  MoveL 5719 to (502.61, 490.4, 12.5) mm, rotated rx 0 ry 90 rz 0 deg; joints [-11.079, -27.597, 111.319, -15.089, -83.075, 50.859]
  Call Extruder(0.203)
  MoveL 5720 to (509.6, 490.4, 12.5) mm, rotated rx 0 ry 90 rz 0 deg; joints [-10.955, -27.463, 110.479, -14.987, -82.389, 51.03]
  Call Extruder(0.176)
  MoveL 5721 to (509.6, 496.43, 12.5) mm, rotated rx 0 ry 90 rz 0 deg; joints [-11.502, -27.439, 110.334, -15.543, -82.29, 51.128]
  Call Extruder(0.056)
  MoveL 5722 to (507.67, 496.44, 12.5) mm, rotated rx 0 ry 90 rz 0 deg; joints [-11.538, -27.477, 110.567, -15.572, -82.478, 51.079]
  Call Extruder(0.062)
  MoveL 5723 to (507.67, 498.58, 12.5) mm, rotated rx 0 ry 90 rz 0 deg; joints [-11.732, -27.468, 110.514, -15.77, -82.442, 51.114]
  Call Extruder(0.010)
  MoveL 5724 to (507.67, 498.93, 12.5) mm, rotated rx 0 ry 90 rz 0 deg; joints [-11.764, -27.467, 110.505, -15.802, -82.436, 51.12]
  Call Extruder(0.007)
  MoveL 5725 to (508.02, 498.93, 12.5) mm, rotated rx 0 ry 90 rz 0 deg; joints [-11.757, -27.46, 110.463, -15.797, -82.402, 51.129]
  Call Extruder(0.036)
  MoveL 5726 to (509.25, 498.93, 12.5) mm, rotated rx 0 ry 90 rz 0 deg; joints [-11.734, -27.436, 110.315, -15.778, -82.282, 51.16]
  Call Extruder(0.010)
  MoveL 5727 to (509.6, 498.93, 12.5) mm, rotated rx 0 ry 90 rz 0 deg; joints [-11.727, -27.429, 110.272, -15.772, -82.248, 51.169]
  Call Extruder(0.007)
  MoveL 5728 to (509.6, 499.28, 12.5) mm, rotated rx 0 ry 90 rz 0 deg; joints [-11.759, -27.427, 110.264, -15.805, -82.242, 51.175]
  Call Extruder(0.016)
  MoveL 5729 to (509.6, 499.84, 12.5) mm, rotated rx 0 ry 90 rz 0 deg; joints [-11.81, -27.425, 110.249, -15.856, -82.232, 51.184]
  Call Extruder(0.010)
  MoveL 5730 to (509.6, 500.19, 12.5) mm, rotated rx 0 ry 90 rz 0 deg; joints [-11.842, -27.423, 110.241, -15.889, -82.226, 51.19]
  Call Extruder(0.007)
  MoveL 5731 to (509.25, 500.19, 12.5) mm, rotated rx 0 ry 90 rz 0 deg; joints [-11.848, -27.43, 110.283, -15.894, -82.26, 51.181]
  Call Extruder(0.036)
  MoveL 5732 to (508.02, 500.19, 12.5) mm, rotated rx 0 ry 90 rz 0 deg; joints [-11.871, -27.455, 110.431, -15.913, -82.38, 51.149]
  Call Extruder(0.010)
  MoveL 5733 to (507.67, 500.19, 12.5) mm, rotated rx 0 ry 90 rz 0 deg; joints [-11.878, -27.462, 110.473, -15.918, -82.414, 51.141]
  Call Extruder(0.007)
  MoveL 5734 to (507.67, 500.54, 12.5) mm, rotated rx 0 ry 90 rz 0 deg; joints [-11.91, -27.46, 110.464, -15.95, -82.408, 51.146]
  Call Extruder(0.062)
  MoveL 5735 to (507.67, 502.67, 12.5) mm, rotated rx 0 ry 90 rz 0 deg; joints [-12.103, -27.451, 110.41, -16.147, -82.371, 51.182]
  Call Extruder(0.056)
  MoveL 5736 to (509.6, 502.68, 12.5) mm, rotated rx 0 ry 90 rz 0 deg; joints [-12.066, -27.413, 110.177, -16.116, -82.183, 51.232]
  Call Extruder(0.202)
  MoveL 5737 to (509.6, 509.6, 12.5) mm, rotated rx 0 ry 90 rz 0 deg; joints [-12.688, -27.382, 109.994, -16.751, -82.06, 51.352]
  Call Extruder(0.559)
  MoveL 5738 to (490.4, 509.6, 12.5) mm, rotated rx 0 ry 90 rz 0 deg; joints [-13.088, -27.741, 112.282, -17.084, -83.918, 50.83]
  MoveL 5739 to (490.4, 490.4, 12.5) mm, rotated rx 0 ry 90 rz 0 deg; joints [-11.303, -27.811, 112.772, -15.278, -84.276, 50.554]
  Call Extruder(0.177)
  MoveL 5740 to (496.5, 490.4, 12.5) mm, rotated rx 0 ry 90 rz 0 deg; joints [-11.19, -27.707, 112.049, -15.182, -83.676, 50.708]
  Call Extruder(0.010)
  MoveL 5741 to (496.85, 490.4, 12.5) mm, rotated rx 0 ry 90 rz 0 deg; joints [-11.184, -27.701, 112.007, -15.177, -83.641, 50.717]
  Call Extruder(0.007)
  MoveL 5742 to (496.85, 490.75, 12.5) mm, rotated rx 0 ry 90 rz 0 deg; joints [-11.216, -27.7, 111.999, -15.209, -83.635, 50.721]
  Call Extruder(0.035)
  MoveL 5743 to (496.84, 491.95, 12.5) mm, rotated rx 0 ry 90 rz 0 deg; joints [-11.327, -27.696, 111.971, -15.322, -83.615, 50.739]
  Call Extruder(0.010)
  MoveL 5744 to (496.84, 492.3, 12.5) mm, rotated rx 0 ry 90 rz 0 deg; joints [-11.36, -27.694, 111.962, -15.355, -83.609, 50.744]
  Call Extruder(0.007)
  MoveL 5745 to (497.19, 492.3, 12.5) mm, rotated rx 0 ry 90 rz 0 deg; joints [-11.353, -27.688, 111.921, -15.349, -83.575, 50.752]
  Call Extruder(0.061)
  MoveL 5746 to (499.3, 492.3, 12.5) mm, rotated rx 0 ry 90 rz 0 deg; joints [-11.314, -27.65, 111.669, -15.316, -83.367, 50.805]
  Call Extruder(0.055)
  MoveL 5747 to (499.3, 490.4, 12.5) mm, rotated rx 0 ry 90 rz 0 deg; joints [-11.139, -27.657, 111.714, -15.139, -83.399, 50.778]
  Call Extruder(0.016)
  MoveL 5748 to (499.84, 490.4, 12.5) mm, rotated rx 0 ry 90 rz 0 deg; joints [-11.129, -27.648, 111.65, -15.131, -83.347, 50.791]
  Call Extruder(0.042)
  MoveL 5749 to (499.84, 492.3, 12.5) mm, rotated rx 0 ry 90 rz 0 deg; joints [-11.304, -27.641, 111.605, -15.308, -83.315, 50.819]
  Call Extruder(0.060)
  MoveL 5750 to (501.91, 492.3, 12.5) mm, rotated rx 0 ry 90 rz 0 deg; joints [-11.266, -27.603, 111.358, -15.276, -83.112, 50.871]
  Call Extruder(0.007)
  MoveL 5751 to (502.26, 492.3, 12.5) mm, rotated rx 0 ry 90 rz 0 deg; joints [-11.26, -27.596, 111.316, -15.271, -83.077, 50.879]
  Set speed (120.0 mm/s)
  MoveL 5752 to (502.26, 491.95, 12.5) mm, rotated rx 0 ry 90 rz 0 deg; joints [-11.228, -27.598, 111.324, -15.238, -83.083, 50.874]
  Set speed (1000.0 mm/s)
  MoveL 5753 to (502.26, 491.9, 12.5) mm, rotated rx 0 ry 90 rz 0 deg; joints [-11.223, -27.598, 111.325, -15.234, -83.084, 50.873]
  Set speed (1000.0 mm/s)
  MoveL 5754 to (502.36, 491.9, 12.5) mm, rotated rx 0 ry 90 rz 0 deg; joints [-11.221, -27.596, 111.313, -15.232, -83.074, 50.876]
  Set speed (1000.0 mm/s)
  MoveL 5755 to (507.28, 499.36, 12.5) mm, rotated rx 0 ry 90 rz 0 deg; joints [-11.811, -27.473, 110.54, -15.848, -82.466, 51.117]
  Set speed (1000.0 mm/s)
  MoveL 5756 to (507.53, 499.61, 12.5) mm, rotated rx 0 ry 90 rz 0 deg; joints [-11.828, -27.467, 110.505, -15.867, -82.438, 51.127]
  Set speed (15.0 mm/s)
  Call Extruder(0.014)
  MoveL 5757 to (507.97, 499.56, 12.5) mm, rotated rx 0 ry 90 rz 0 deg; joints [-11.815, -27.458, 110.452, -15.855, -82.396, 51.138]
  Call Extruder(0.030)
  MoveL 5758 to (508.96, 499.56, 12.5) mm, rotated rx 0 ry 90 rz 0 deg; joints [-11.796, -27.439, 110.333, -15.84, -82.299, 51.163]
  Call Extruder(0.011)
  MoveL 5759 to (509.21, 499.31, 12.5) mm, rotated rx 0 ry 90 rz 0 deg; joints [-11.77, -27.435, 110.309, -15.814, -82.279, 51.165]
  Set speed (120.0 mm/s)
  MoveL 5760 to (508.9, 499.63, 12.5) mm, rotated rx 0 ry 90 rz 0 deg; joints [-11.804, -27.44, 110.339, -15.848, -82.304, 51.163]
  Set speed (1000.0 mm/s)
  MoveL 5761 to (490.68, 490.68, 12.5) mm, rotated rx 0 ry 90 rz 0 deg; joints [-11.324, -27.805, 112.732, -15.3, -84.244, 50.565]
  Set speed (1000.0 mm/s)
  MoveL 5762 to (490.68, 490.68, 12.6) mm, rotated rx 0 ry 90 rz 0 deg; joints [-11.324, -27.816, 112.737, -15.3, -84.238, 50.567]
  Set speed (30.0 mm/s)
  Call Extruder(0.767)
  MoveL 5763 to (509.32, 509.32, 12.6) mm, rotated rx 0 ry 90 rz 0 deg; joints [-12.669, -27.4, 110.041, -16.73, -82.087, 51.341]
  MoveL 5764 to (509.44, 509.44, 12.6) mm, rotated rx 0 ry 90 rz 0 deg; joints [-12.677, -27.397, 110.023, -16.739, -82.073, 51.347]
  Set speed (120.0 mm/s)
  MoveL 5765 to (507.39, 502.51, 12.6) mm, rotated rx 0 ry 90 rz 0 deg; joints [-12.094, -27.468, 110.453, -16.137, -82.396, 51.173]
  Set speed (30.0 mm/s)
  Call Extruder(0.280)
  MoveL 5766 to (500.58, 509.32, 12.6) mm, rotated rx 0 ry 90 rz 0 deg; joints [-12.847, -27.57, 111.088, -16.877, -82.932, 51.106]
  Set speed (120.0 mm/s)
  MoveL 5767 to (499.42, 509.32, 12.6) mm, rotated rx 0 ry 90 rz 0 deg; joints [-12.872, -27.592, 111.226, -16.897, -83.044, 51.075]
  Set speed (30.0 mm/s)
  Call Extruder(0.360)
  MoveL 5768 to (490.68, 500.58, 12.6) mm, rotated rx 0 ry 90 rz 0 deg; joints [-12.247, -27.781, 112.493, -16.233, -84.059, 50.705]
  Set speed (120.0 mm/s)
  MoveL 5769 to (490.68, 499.42, 12.6) mm, rotated rx 0 ry 90 rz 0 deg; joints [-12.139, -27.786, 112.523, -16.124, -84.081, 50.688]
  Set speed (30.0 mm/s)
  Call Extruder(0.282)
  MoveL 5770 to (497.52, 492.58, 12.6) mm, rotated rx 0 ry 90 rz 0 deg; joints [-11.373, -27.692, 111.88, -15.37, -83.533, 50.766]
  MoveL 5771 to (497.64, 492.46, 12.6) mm, rotated rx 0 ry 90 rz 0 deg; joints [-11.359, -27.69, 111.869, -15.357, -83.523, 50.767]
  Set speed (120.0 mm/s)
  MoveL 5772 to (502.48, 492.58, 12.6) mm, rotated rx 0 ry 90 rz 0 deg; joints [-11.281, -27.602, 111.288, -15.294, -83.046, 50.89]
  Set speed (30.0 mm/s)
  Call Extruder(0.202)
  MoveL 5773 to (507.39, 497.49, 12.6) mm, rotated rx 0 ry 90 rz 0 deg; joints [-11.639, -27.489, 110.58, -15.674, -82.483, 51.091]
  MoveL 5774 to (507.51, 497.61, 12.6) mm, rotated rx 0 ry 90 rz 0 deg; joints [-11.647, -27.486, 110.562, -15.683, -82.469, 51.096]
  Set speed (120.0 mm/s)
  MoveL 5775 to (509.32, 490.68, 12.6) mm, rotated rx 0 ry 90 rz 0 deg; joints [-10.985, -27.478, 110.511, -15.017, -82.407, 51.029]
  Set speed (30.0 mm/s)
  Call Extruder(0.767)
  MoveL 5776 to (490.68, 509.32, 12.6) mm, rotated rx 0 ry 90 rz 0 deg; joints [-13.056, -27.748, 112.262, -17.053, -83.891, 50.835]
  MoveL 5777 to (490.56, 509.44, 12.6) mm, rotated rx 0 ry 90 rz 0 deg; joints [-13.07, -27.75, 112.273, -17.067, -83.901, 50.833]
  Set speed (120.0 mm/s)
  MoveL 5778 to (496.72, 492.37, 12.6) mm, rotated rx 0 ry 90 rz 0 deg; joints [-11.369, -27.707, 111.981, -15.363, -83.615, 50.743]
  Set speed (1000.0 mm/s)
  MoveL 5779 to (496.79, 492.3, 12.6) mm, rotated rx 0 ry 90 rz 0 deg; joints [-11.361, -27.706, 111.974, -15.356, -83.609, 50.744]
  Set speed (15.0 mm/s)
  Call Extruder(0.072)
  MoveL 5780 to (499.25, 492.3, 12.6) mm, rotated rx 0 ry 90 rz 0 deg; joints [-11.315, -27.662, 111.681, -15.317, -83.368, 50.806]
  Call Extruder(0.055)
  MoveL 5781 to (499.25, 490.4, 12.6) mm, rotated rx 0 ry 90 rz 0 deg; joints [-11.14, -27.669, 111.726, -15.14, -83.4, 50.778]
  Call Extruder(0.019)
  MoveL 5782 to (499.9, 490.4, 12.6) mm, rotated rx 0 ry 90 rz 0 deg; joints [-11.128, -27.657, 111.648, -15.13, -83.336, 50.794]
  Call Extruder(0.052)
  MoveL 5783 to (499.9, 492.3, 12.6) mm, rotated rx 0 ry 90 rz 0 deg; joints [-11.303, -27.65, 111.603, -15.307, -83.303, 50.822]
  Call Extruder(0.060)
  MoveL 5784 to (501.97, 492.3, 12.6) mm, rotated rx 0 ry 90 rz 0 deg; joints [-11.265, -27.612, 111.355, -15.276, -83.1, 50.874]
  Call Extruder(0.010)
  MoveL 5785 to (502.32, 492.3, 12.6) mm, rotated rx 0 ry 90 rz 0 deg; joints [-11.259, -27.606, 111.313, -15.27, -83.066, 50.882]
  Call Extruder(0.007)
  MoveL 5786 to (502.32, 491.95, 12.6) mm, rotated rx 0 ry 90 rz 0 deg; joints [-11.227, -27.607, 111.322, -15.238, -83.072, 50.877]
  Call Extruder(0.035)
  MoveL 5787 to (502.32, 490.75, 12.6) mm, rotated rx 0 ry 90 rz 0 deg; joints [-11.116, -27.611, 111.35, -15.126, -83.092, 50.859]
  Call Extruder(0.010)
  MoveL 5788 to (502.32, 490.4, 12.6) mm, rotated rx 0 ry 90 rz 0 deg; joints [-11.084, -27.613, 111.358, -15.094, -83.098, 50.854]
  Call Extruder(0.007)
  MoveL 5789 to (502.67, 490.4, 12.6) mm, rotated rx 0 ry 90 rz 0 deg; joints [-11.078, -27.606, 111.317, -15.088, -83.063, 50.862]
  Call Extruder(0.202)
  MoveL 5790 to (509.6, 490.4, 12.6) mm, rotated rx 0 ry 90 rz 0 deg; joints [-10.955, -27.473, 110.484, -14.987, -82.384, 51.032]
  Call Extruder(0.174)
  MoveL 5791 to (509.6, 496.37, 12.6) mm, rotated rx 0 ry 90 rz 0 deg; joints [-11.496, -27.45, 110.341, -15.538, -82.286, 51.128]
  Call Extruder(0.056)
  MoveL 5792 to (507.67, 496.38, 12.6) mm, rotated rx 0 ry 90 rz 0 deg; joints [-11.532, -27.488, 110.573, -15.567, -82.474, 51.08]
  Call Extruder(0.073)
  MoveL 5793 to (507.67, 498.87, 12.6) mm, rotated rx 0 ry 90 rz 0 deg; joints [-11.759, -27.478, 110.511, -15.797, -82.432, 51.12]
  Call Extruder(0.056)
  MoveL 5794 to (509.6, 498.87, 12.6) mm, rotated rx 0 ry 90 rz 0 deg; joints [-11.722, -27.439, 110.279, -15.767, -82.244, 51.169]
  Call Extruder(0.030)
  MoveL 5795 to (509.6, 499.9, 12.6) mm, rotated rx 0 ry 90 rz 0 deg; joints [-11.815, -27.435, 110.253, -15.862, -82.226, 51.186]
  Call Extruder(0.010)
  MoveL 5796 to (509.6, 500.25, 12.6) mm, rotated rx 0 ry 90 rz 0 deg; joints [-11.847, -27.434, 110.244, -15.894, -82.22, 51.192]
  Call Extruder(0.007)
  MoveL 5797 to (509.25, 500.25, 12.6) mm, rotated rx 0 ry 90 rz 0 deg; joints [-11.853, -27.441, 110.286, -15.899, -82.254, 51.183]
  Call Extruder(0.036)
  MoveL 5798 to (508.02, 500.25, 12.6) mm, rotated rx 0 ry 90 rz 0 deg; joints [-11.876, -27.465, 110.435, -15.918, -82.374, 51.152]
  Call Extruder(0.010)
  MoveL 5799 to (507.67, 500.25, 12.6) mm, rotated rx 0 ry 90 rz 0 deg; joints [-11.883, -27.472, 110.477, -15.924, -82.408, 51.143]
  Call Extruder(0.007)
  MoveL 5800 to (507.67, 500.6, 12.6) mm, rotated rx 0 ry 90 rz 0 deg; joints [-11.915, -27.471, 110.468, -15.956, -82.402, 51.149]
  Call Extruder(0.062)
  MoveL 5801 to (507.67, 502.73, 12.6) mm, rotated rx 0 ry 90 rz 0 deg; joints [-12.108, -27.462, 110.414, -16.152, -82.365, 51.184]
  Call Extruder(0.056)
  MoveL 5802 to (509.6, 502.73, 12.6) mm, rotated rx 0 ry 90 rz 0 deg; joints [-12.071, -27.423, 110.181, -16.122, -82.177, 51.234]
  Call Extruder(0.200)
  MoveL 5803 to (509.6, 509.6, 12.6) mm, rotated rx 0 ry 90 rz 0 deg; joints [-12.688, -27.393, 109.999, -16.751, -82.055, 51.354]
  Call Extruder(0.559)
  MoveL 5804 to (490.4, 509.6, 12.6) mm, rotated rx 0 ry 90 rz 0 deg; joints [-13.088, -27.752, 112.287, -17.084, -83.913, 50.831]
  MoveL 5805 to (490.4, 490.4, 12.6) mm, rotated rx 0 ry 90 rz 0 deg; joints [-11.303, -27.821, 112.777, -15.278, -84.271, 50.556]
  Call Extruder(0.176)
  MoveL 5806 to (496.44, 490.4, 12.6) mm, rotated rx 0 ry 90 rz 0 deg; joints [-11.191, -27.719, 112.061, -15.183, -83.676, 50.708]
  Call Extruder(0.010)
  MoveL 5807 to (496.79, 490.4, 12.6) mm, rotated rx 0 ry 90 rz 0 deg; joints [-11.185, -27.713, 112.019, -15.178, -83.642, 50.717]
  Call Extruder(0.007)
  MoveL 5808 to (496.79, 490.75, 12.6) mm, rotated rx 0 ry 90 rz 0 deg; joints [-11.217, -27.711, 112.011, -15.21, -83.636, 50.722]
  Call Extruder(0.045)
  MoveL 5809 to (496.79, 492.3, 12.6) mm, rotated rx 0 ry 90 rz 0 deg; joints [-11.361, -27.706, 111.974, -15.356, -83.609, 50.744]
  Set speed (120.0 mm/s)
  MoveL 5810 to (497.19, 492.3, 12.6) mm, rotated rx 0 ry 90 rz 0 deg; joints [-11.353, -27.699, 111.926, -15.349, -83.57, 50.754]
  Set speed (1000.0 mm/s)
  MoveL 5811 to (497.19, 492.4, 12.6) mm, rotated rx 0 ry 90 rz 0 deg; joints [-11.363, -27.699, 111.924, -15.359, -83.568, 50.755]
  Set speed (1000.0 mm/s)
  MoveL 5812 to (507.28, 499.5, 12.6) mm, rotated rx 0 ry 90 rz 0 deg; joints [-11.822, -27.483, 110.542, -15.86, -82.459, 51.121]
  Set speed (15.0 mm/s)
  Call Extruder(0.006)
  MoveL 5813 to (507.58, 499.2, 12.6) mm, rotated rx 0 ry 90 rz 0 deg; joints [-11.79, -27.478, 110.514, -15.829, -82.435, 51.123]
  Set speed (120.0 mm/s)
  MoveL 5814 to (508.07, 499.2, 12.6) mm, rotated rx 0 ry 90 rz 0 deg; joints [-11.781, -27.468, 110.455, -15.821, -82.387, 51.136]
  Set speed (15.0 mm/s)
  Call Extruder(0.015)
  MoveL 5815 to (507.36, 499.91, 12.6) mm, rotated rx 0 ry 90 rz 0 deg; joints [-11.859, -27.48, 110.522, -15.898, -82.444, 51.13]
  Set speed (120.0 mm/s)
  MoveL 5816 to (507.85, 499.92, 12.6) mm, rotated rx 0 ry 90 rz 0 deg; joints [-11.85, -27.47, 110.463, -15.89, -82.396, 51.142]
  Set speed (15.0 mm/s)
  Call Extruder(0.015)
  MoveL 5817 to (508.57, 499.2, 12.6) mm, rotated rx 0 ry 90 rz 0 deg; joints [-11.771, -27.459, 110.395, -15.813, -82.339, 51.149]
  Set speed (120.0 mm/s)
  MoveL 5818 to (509.06, 499.2, 12.6) mm, rotated rx 0 ry 90 rz 0 deg; joints [-11.762, -27.449, 110.335, -15.806, -82.29, 51.161]
  Set speed (15.0 mm/s)
  Call Extruder(0.015)
  MoveL 5819 to (508.35, 499.92, 12.6) mm, rotated rx 0 ry 90 rz 0 deg; joints [-11.84, -27.46, 110.404, -15.883, -82.348, 51.155]
  Set speed (120.0 mm/s)
  MoveL 5820 to (508.84, 499.92, 12.6) mm, rotated rx 0 ry 90 rz 0 deg; joints [-11.831, -27.45, 110.344, -15.875, -82.3, 51.167]
  Set speed (15.0 mm/s)
  Call Extruder(0.009)
  MoveL 5821 to (509.27, 499.49, 12.6) mm, rotated rx 0 ry 90 rz 0 deg; joints [-11.784, -27.443, 110.303, -15.829, -82.266, 51.171]
  Set speed (120.0 mm/s)
  MoveL 5822 to (508.9, 499.57, 12.6) mm, rotated rx 0 ry 90 rz 0 deg; joints [-11.799, -27.45, 110.346, -15.842, -82.3, 51.163]
  Set speed (1000.0 mm/s)
  MoveL 5823 to (490.68, 490.68, 12.6) mm, rotated rx 0 ry 90 rz 0 deg; joints [-11.324, -27.816, 112.737, -15.3, -84.238, 50.567]
  Set speed (1000.0 mm/s)
  MoveL 5824 to (490.68, 490.68, 12.7) mm, rotated rx 0 ry 90 rz 0 deg; joints [-11.324, -27.826, 112.742, -15.3, -84.233, 50.568]
  Set speed (30.0 mm/s)
  Call Extruder(0.767)
  MoveL 5825 to (509.32, 509.32, 12.7) mm, rotated rx 0 ry 90 rz 0 deg; joints [-12.669, -27.41, 110.046, -16.73, -82.082, 51.343]
  MoveL 5826 to (509.44, 509.44, 12.7) mm, rotated rx 0 ry 90 rz 0 deg; joints [-12.677, -27.407, 110.028, -16.739, -82.068, 51.348]
  Set speed (120.0 mm/s)
  MoveL 5827 to (507.38, 502.51, 12.7) mm, rotated rx 0 ry 90 rz 0 deg; joints [-12.094, -27.479, 110.458, -16.137, -82.391, 51.175]
  Set speed (30.0 mm/s)
  Call Extruder(0.280)
  MoveL 5828 to (500.58, 509.32, 12.7) mm, rotated rx 0 ry 90 rz 0 deg; joints [-12.847, -27.581, 111.093, -16.877, -82.927, 51.108]
  Set speed (120.0 mm/s)
  MoveL 5829 to (499.42, 509.32, 12.7) mm, rotated rx 0 ry 90 rz 0 deg; joints [-12.872, -27.603, 111.231, -16.897, -83.039, 51.077]
  Set speed (30.0 mm/s)
  Call Extruder(0.360)
  MoveL 5830 to (490.68, 500.58, 12.7) mm, rotated rx 0 ry 90 rz 0 deg; joints [-12.247, -27.792, 112.498, -16.234, -84.054, 50.706]
  Set speed (120.0 mm/s)
  MoveL 5831 to (490.68, 499.42, 12.7) mm, rotated rx 0 ry 90 rz 0 deg; joints [-12.139, -27.796, 112.528, -16.124, -84.076, 50.689]
  Set speed (30.0 mm/s)
  Call Extruder(0.281)
  MoveL 5832 to (497.52, 492.58, 12.7) mm, rotated rx 0 ry 90 rz 0 deg; joints [-11.373, -27.703, 111.886, -15.371, -83.527, 50.768]
  MoveL 5833 to (497.64, 492.46, 12.7) mm, rotated rx 0 ry 90 rz 0 deg; joints [-11.359, -27.701, 111.874, -15.357, -83.517, 50.769]
  Set speed (120.0 mm/s)
  MoveL 5834 to (502.48, 492.58, 12.7) mm, rotated rx 0 ry 90 rz 0 deg; joints [-11.282, -27.612, 111.293, -15.294, -83.041, 50.892]
  Set speed (30.0 mm/s)
  Call Extruder(0.202)
  MoveL 5835 to (507.39, 497.49, 12.7) mm, rotated rx 0 ry 90 rz 0 deg; joints [-11.639, -27.499, 110.585, -15.674, -82.478, 51.092]
  MoveL 5836 to (507.51, 497.61, 12.7) mm, rotated rx 0 ry 90 rz 0 deg; joints [-11.647, -27.496, 110.567, -15.683, -82.464, 51.097]
  Set speed (120.0 mm/s)
  MoveL 5837 to (508.99, 499.09, 12.7) mm, rotated rx 0 ry 90 rz 0 deg; joints [-11.754, -27.461, 110.352, -15.797, -82.294, 51.159]
  Set speed (30.0 mm/s)
  Call Extruder(0.013)
  MoveL 5838 to (509.32, 499.42, 12.7) mm, rotated rx 0 ry 90 rz 0 deg; joints [-11.777, -27.453, 110.304, -15.822, -82.257, 51.173]
  Set speed (120.0 mm/s)
  MoveL 5839 to (507.64, 498.84, 12.7) mm, rotated rx 0 ry 90 rz 0 deg; joints [-11.756, -27.489, 110.521, -15.795, -82.43, 51.121]
  Set speed (1000.0 mm/s)
  MoveL 5840 to (507.64, 496.29, 12.7) mm, rotated rx 0 ry 90 rz 0 deg; joints [-11.525, -27.499, 110.584, -15.559, -82.473, 51.079]
  Set speed (1000.0 mm/s)
  MoveL 5841 to (509.32, 490.68, 12.7) mm, rotated rx 0 ry 90 rz 0 deg; joints [-10.985, -27.488, 110.516, -15.017, -82.402, 51.031]
  Set speed (30.0 mm/s)
  Call Extruder(0.767)
  MoveL 5842 to (490.68, 509.32, 12.7) mm, rotated rx 0 ry 90 rz 0 deg; joints [-13.056, -27.759, 112.267, -17.053, -83.886, 50.836]
  MoveL 5843 to (490.56, 509.44, 12.7) mm, rotated rx 0 ry 90 rz 0 deg; joints [-13.07, -27.76, 112.278, -17.067, -83.895, 50.835]
  Set speed (120.0 mm/s)
  MoveL 5844 to (502.46, 492.37, 12.7) mm, rotated rx 0 ry 90 rz 0 deg; joints [-11.263, -27.613, 111.301, -15.275, -83.046, 50.888]
  Set speed (1000.0 mm/s)
  MoveL 5845 to (502.39, 492.3, 12.7) mm, rotated rx 0 ry 90 rz 0 deg; joints [-11.257, -27.615, 111.311, -15.269, -83.054, 50.885]
  Set speed (15.0 mm/s)
  Call Extruder(0.010)
  MoveL 5846 to (502.39, 491.95, 12.7) mm, rotated rx 0 ry 90 rz 0 deg; joints [-11.225, -27.616, 111.319, -15.237, -83.06, 50.88]
  Call Extruder(0.035)
  MoveL 5847 to (502.39, 490.75, 12.7) mm, rotated rx 0 ry 90 rz 0 deg; joints [-11.115, -27.621, 111.348, -15.125, -83.08, 50.862]
  Call Extruder(0.010)
  MoveL 5848 to (502.39, 490.4, 12.7) mm, rotated rx 0 ry 90 rz 0 deg; joints [-11.083, -27.622, 111.356, -15.093, -83.086, 50.857]
  Call Extruder(0.007)
  MoveL 5849 to (502.74, 490.4, 12.7) mm, rotated rx 0 ry 90 rz 0 deg; joints [-11.077, -27.616, 111.314, -15.088, -83.052, 50.865]
  Call Extruder(0.200)
  MoveL 5850 to (509.6, 490.4, 12.7) mm, rotated rx 0 ry 90 rz 0 deg; joints [-10.955, -27.484, 110.489, -14.988, -82.378, 51.033]
  Call Extruder(0.172)
  MoveL 5851 to (509.6, 496.31, 12.7) mm, rotated rx 0 ry 90 rz 0 deg; joints [-11.491, -27.46, 110.347, -15.532, -82.282, 51.128]
  Call Extruder(0.056)
  MoveL 5852 to (507.67, 496.31, 12.7) mm, rotated rx 0 ry 90 rz 0 deg; joints [-11.527, -27.499, 110.58, -15.562, -82.47, 51.08]
  Call Extruder(0.062)
  MoveL 5853 to (507.67, 498.46, 12.7) mm, rotated rx 0 ry 90 rz 0 deg; joints [-11.722, -27.49, 110.527, -15.759, -82.434, 51.115]
  Call Extruder(0.010)
  MoveL 5854 to (507.67, 498.81, 12.7) mm, rotated rx 0 ry 90 rz 0 deg; joints [-11.753, -27.488, 110.518, -15.792, -82.428, 51.121]
  Call Extruder(0.007)
  MoveL 5855 to (508.02, 498.81, 12.7) mm, rotated rx 0 ry 90 rz 0 deg; joints [-11.747, -27.482, 110.476, -15.786, -82.394, 51.13]
  Call Extruder(0.036)
  MoveL 5856 to (509.25, 498.81, 12.7) mm, rotated rx 0 ry 90 rz 0 deg; joints [-11.723, -27.457, 110.328, -15.767, -82.274, 51.161]
  Call Extruder(0.010)
  MoveL 5857 to (509.6, 498.81, 12.7) mm, rotated rx 0 ry 90 rz 0 deg; joints [-11.717, -27.45, 110.286, -15.762, -82.24, 51.17]
  Call Extruder(0.007)
  MoveL 5858 to (509.6, 499.16, 12.7) mm, rotated rx 0 ry 90 rz 0 deg; joints [-11.749, -27.449, 110.277, -15.794, -82.234, 51.176]
  Call Extruder(0.023)
  MoveL 5859 to (509.6, 499.95, 12.7) mm, rotated rx 0 ry 90 rz 0 deg; joints [-11.82, -27.445, 110.257, -15.867, -82.22, 51.189]
  Call Extruder(0.010)
  MoveL 5860 to (509.6, 500.3, 12.7) mm, rotated rx 0 ry 90 rz 0 deg; joints [-11.852, -27.444, 110.248, -15.899, -82.214, 51.195]
  Call Extruder(0.007)
  MoveL 5861 to (509.25, 500.3, 12.7) mm, rotated rx 0 ry 90 rz 0 deg; joints [-11.858, -27.451, 110.29, -15.905, -82.248, 51.186]
  Call Extruder(0.036)
  MoveL 5862 to (508.02, 500.3, 12.7) mm, rotated rx 0 ry 90 rz 0 deg; joints [-11.882, -27.475, 110.439, -15.924, -82.368, 51.154]
  Call Extruder(0.010)
  MoveL 5863 to (507.67, 500.3, 12.7) mm, rotated rx 0 ry 90 rz 0 deg; joints [-11.888, -27.482, 110.481, -15.929, -82.402, 51.145]
  Call Extruder(0.007)
  MoveL 5864 to (507.67, 500.65, 12.7) mm, rotated rx 0 ry 90 rz 0 deg; joints [-11.92, -27.481, 110.472, -15.961, -82.396, 51.151]
  Call Extruder(0.062)
  MoveL 5865 to (507.67, 502.79, 12.7) mm, rotated rx 0 ry 90 rz 0 deg; joints [-12.113, -27.472, 110.417, -16.157, -82.359, 51.187]
  Call Extruder(0.056)
  MoveL 5866 to (509.6, 502.79, 12.7) mm, rotated rx 0 ry 90 rz 0 deg; joints [-12.076, -27.433, 110.185, -16.127, -82.171, 51.237]
  Call Extruder(0.198)
  MoveL 5867 to (509.6, 509.6, 12.7) mm, rotated rx 0 ry 90 rz 0 deg; joints [-12.688, -27.403, 110.004, -16.751, -82.049, 51.355]
  Call Extruder(0.559)
  MoveL 5868 to (490.4, 509.6, 12.7) mm, rotated rx 0 ry 90 rz 0 deg; joints [-13.088, -27.762, 112.292, -17.084, -83.907, 50.833]
  MoveL 5869 to (490.4, 490.4, 12.7) mm, rotated rx 0 ry 90 rz 0 deg; joints [-11.303, -27.832, 112.782, -15.279, -84.265, 50.557]
  Call Extruder(0.174)
  MoveL 5870 to (496.38, 490.4, 12.7) mm, rotated rx 0 ry 90 rz 0 deg; joints [-11.192, -27.73, 112.072, -15.184, -83.676, 50.708]
  Call Extruder(0.010)
  MoveL 5871 to (496.73, 490.4, 12.7) mm, rotated rx 0 ry 90 rz 0 deg; joints [-11.186, -27.724, 112.031, -15.179, -83.642, 50.717]
  Call Extruder(0.007)
  MoveL 5872 to (496.73, 490.75, 12.7) mm, rotated rx 0 ry 90 rz 0 deg; joints [-11.218, -27.723, 112.023, -15.211, -83.636, 50.722]
  Call Extruder(0.035)
  MoveL 5873 to (496.73, 491.95, 12.7) mm, rotated rx 0 ry 90 rz 0 deg; joints [-11.329, -27.719, 111.994, -15.324, -83.615, 50.739]
  Call Extruder(0.010)
  MoveL 5874 to (496.73, 492.3, 12.7) mm, rotated rx 0 ry 90 rz 0 deg; joints [-11.362, -27.718, 111.986, -15.357, -83.609, 50.744]
  Call Extruder(0.007)
  MoveL 5875 to (497.08, 492.3, 12.7) mm, rotated rx 0 ry 90 rz 0 deg; joints [-11.355, -27.711, 111.944, -15.351, -83.575, 50.753]
  Call Extruder(0.061)
  MoveL 5876 to (499.19, 492.3, 12.7) mm, rotated rx 0 ry 90 rz 0 deg; joints [-11.316, -27.674, 111.693, -15.318, -83.368, 50.806]
  Call Extruder(0.055)
  MoveL 5877 to (499.19, 490.4, 12.7) mm, rotated rx 0 ry 90 rz 0 deg; joints [-11.141, -27.68, 111.738, -15.141, -83.4, 50.778]
  Call Extruder(0.022)
  MoveL 5878 to (499.96, 490.4, 12.7) mm, rotated rx 0 ry 90 rz 0 deg; joints [-11.127, -27.666, 111.646, -15.129, -83.324, 50.797]
  Call Extruder(0.055)
  MoveL 5879 to (499.97, 492.3, 12.7) mm, rotated rx 0 ry 90 rz 0 deg; joints [-11.302, -27.66, 111.6, -15.307, -83.292, 50.825]
  Call Extruder(0.060)
  MoveL 5880 to (502.04, 492.3, 12.7) mm, rotated rx 0 ry 90 rz 0 deg; joints [-11.264, -27.622, 111.353, -15.275, -83.089, 50.877]
  Call Extruder(0.007)
  MoveL 5881 to (502.39, 492.3, 12.7) mm, rotated rx 0 ry 90 rz 0 deg; joints [-11.257, -27.615, 111.311, -15.269, -83.054, 50.885]
  Set speed (120.0 mm/s)
  MoveL 5882 to (502.39, 491.95, 12.7) mm, rotated rx 0 ry 90 rz 0 deg; joints [-11.225, -27.616, 111.319, -15.237, -83.06, 50.88]
  Set speed (1000.0 mm/s)
  MoveL 5883 to (502.39, 491.9, 12.7) mm, rotated rx 0 ry 90 rz 0 deg; joints [-11.221, -27.617, 111.32, -15.232, -83.061, 50.879]
  Set speed (1000.0 mm/s)
  MoveL 5884 to (502.49, 491.9, 12.7) mm, rotated rx 0 ry 90 rz 0 deg; joints [-11.219, -27.615, 111.308, -15.231, -83.051, 50.882]
  Set speed (1000.0 mm/s)
  MoveL 5885 to (499.94, 492.33, 12.7) mm, rotated rx 0 ry 90 rz 0 deg; joints [-11.305, -27.66, 111.603, -15.31, -83.294, 50.825]
  Set speed (1000.0 mm/s)
  MoveL 5886 to (499.58, 491.66, 12.7) mm, rotated rx 0 ry 90 rz 0 deg; joints [-11.25, -27.669, 111.662, -15.253, -83.341, 50.806]
  Set speed (15.0 mm/s)
  Call Extruder(0.002)
  MoveL 5887 to (499.58, 491.16, 12.7) mm, rotated rx 0 ry 90 rz 0 deg; joints [-11.204, -27.671, 111.674, -15.206, -83.349, 50.798]
  Call Extruder(0.007)
  MoveL 5888 to (499.57, 492.64, 12.7) mm, rotated rx 0 ry 90 rz 0 deg; joints [-11.34, -27.666, 111.64, -15.344, -83.325, 50.82]
  Set speed (120.0 mm/s)
  MoveL 5889 to (499.69, 492.8, 12.7) mm, rotated rx 0 ry 90 rz 0 deg; joints [-11.353, -27.663, 111.622, -15.357, -83.311, 50.825]
  Set speed (1000.0 mm/s)
  MoveL 5890 to (497, 492.38, 12.7) mm, rotated rx 0 ry 90 rz 0 deg; joints [-11.364, -27.712, 111.952, -15.36, -83.582, 50.752]
  Set speed (1000.0 mm/s)
  MoveL 5891 to (490.68, 490.68, 12.7) mm, rotated rx 0 ry 90 rz 0 deg; joints [-11.324, -27.826, 112.742, -15.3, -84.233, 50.568]
  Set speed (1000.0 mm/s)
  MoveL 5892 to (490.68, 490.68, 12.8) mm, rotated rx 0 ry 90 rz 0 deg; joints [-11.324, -27.837, 112.748, -15.301, -84.228, 50.57]
  Set speed (30.0 mm/s)
  Call Extruder(0.767)
  MoveL 5893 to (509.32, 509.32, 12.8) mm, rotated rx 0 ry 90 rz 0 deg; joints [-12.669, -27.421, 110.051, -16.73, -82.077, 51.344]
  MoveL 5894 to (509.44, 509.44, 12.8) mm, rotated rx 0 ry 90 rz 0 deg; joints [-12.677, -27.417, 110.033, -16.739, -82.062, 51.35]
  Set speed (120.0 mm/s)
  MoveL 5895 to (507.38, 502.51, 12.8) mm, rotated rx 0 ry 90 rz 0 deg; joints [-12.094, -27.489, 110.463, -16.137, -82.386, 51.176]
  Set speed (30.0 mm/s)
  Call Extruder(0.280)
  MoveL 5896 to (500.58, 509.32, 12.8) mm, rotated rx 0 ry 90 rz 0 deg; joints [-12.847, -27.591, 111.098, -16.877, -82.922, 51.11]
  Set speed (120.0 mm/s)
  MoveL 5897 to (499.42, 509.32, 12.8) mm, rotated rx 0 ry 90 rz 0 deg; joints [-12.872, -27.613, 111.236, -16.897, -83.034, 51.078]
  Set speed (30.0 mm/s)
  Call Extruder(0.360)
  MoveL 5898 to (490.68, 500.58, 12.8) mm, rotated rx 0 ry 90 rz 0 deg; joints [-12.247, -27.803, 112.504, -16.234, -84.049, 50.708]
  Set speed (120.0 mm/s)
  MoveL 5899 to (490.68, 499.42, 12.8) mm, rotated rx 0 ry 90 rz 0 deg; joints [-12.139, -27.807, 112.533, -16.125, -84.07, 50.691]
  Set speed (30.0 mm/s)
  Call Extruder(0.282)
  MoveL 5900 to (497.52, 492.58, 12.8) mm, rotated rx 0 ry 90 rz 0 deg; joints [-11.373, -27.713, 111.891, -15.371, -83.522, 50.769]
  MoveL 5901 to (497.64, 492.46, 12.8) mm, rotated rx 0 ry 90 rz 0 deg; joints [-11.359, -27.711, 111.879, -15.357, -83.512, 50.77]
  Set speed (120.0 mm/s)
  MoveL 5902 to (502.48, 492.58, 12.8) mm, rotated rx 0 ry 90 rz 0 deg; joints [-11.281, -27.623, 111.298, -15.294, -83.036, 50.893]
  Set speed (30.0 mm/s)
  Call Extruder(0.202)
  MoveL 5903 to (507.39, 497.49, 12.8) mm, rotated rx 0 ry 90 rz 0 deg; joints [-11.639, -27.51, 110.59, -15.674, -82.473, 51.094]
  MoveL 5904 to (507.51, 497.61, 12.8) mm, rotated rx 0 ry 90 rz 0 deg; joints [-11.647, -27.507, 110.572, -15.684, -82.458, 51.099]
  Set speed (120.0 mm/s)
  MoveL 5905 to (508.93, 499.03, 12.8) mm, rotated rx 0 ry 90 rz 0 deg; joints [-11.749, -27.473, 110.366, -15.793, -82.296, 51.158]
  Set speed (30.0 mm/s)
  Call Extruder(0.016)
  MoveL 5906 to (509.32, 499.42, 12.8) mm, rotated rx 0 ry 90 rz 0 deg; joints [-11.777, -27.464, 110.309, -15.823, -82.251, 51.174]
  Set speed (120.0 mm/s)
  MoveL 5907 to (507.64, 498.78, 12.8) mm, rotated rx 0 ry 90 rz 0 deg; joints [-11.751, -27.5, 110.527, -15.789, -82.426, 51.121]
  Set speed (1000.0 mm/s)
  MoveL 5908 to (507.64, 496.23, 12.8) mm, rotated rx 0 ry 90 rz 0 deg; joints [-11.519, -27.51, 110.591, -15.554, -82.469, 51.079]
  Set speed (1000.0 mm/s)
  MoveL 5909 to (509.32, 490.68, 12.8) mm, rotated rx 0 ry 90 rz 0 deg; joints [-10.985, -27.499, 110.521, -15.018, -82.396, 51.032]
  Set speed (30.0 mm/s)
  Call Extruder(0.767)
  MoveL 5910 to (490.68, 509.32, 12.8) mm, rotated rx 0 ry 90 rz 0 deg; joints [-13.056, -27.769, 112.272, -17.053, -83.881, 50.838]
  MoveL 5911 to (490.56, 509.44, 12.8) mm, rotated rx 0 ry 90 rz 0 deg; joints [-13.07, -27.771, 112.283, -17.067, -83.89, 50.837]
  Set speed (120.0 mm/s)
  MoveL 5912 to (502.52, 492.37, 12.8) mm, rotated rx 0 ry 90 rz 0 deg; joints [-11.261, -27.623, 111.298, -15.274, -83.035, 50.891]
  Set speed (1000.0 mm/s)
  MoveL 5913 to (502.45, 492.3, 12.8) mm, rotated rx 0 ry 90 rz 0 deg; joints [-11.256, -27.624, 111.308, -15.269, -83.043, 50.888]
  Set speed (15.0 mm/s)
  Call Extruder(0.010)
  MoveL 5914 to (502.45, 491.95, 12.8) mm, rotated rx 0 ry 90 rz 0 deg; joints [-11.224, -27.626, 111.317, -15.236, -83.049, 50.883]
  Call Extruder(0.035)
  MoveL 5915 to (502.45, 490.75, 12.8) mm, rotated rx 0 ry 90 rz 0 deg; joints [-11.114, -27.63, 111.345, -15.125, -83.069, 50.865]
  Call Extruder(0.010)
  MoveL 5916 to (502.45, 490.4, 12.8) mm, rotated rx 0 ry 90 rz 0 deg; joints [-11.082, -27.631, 111.353, -15.092, -83.075, 50.86]
  Call Extruder(0.007)
  MoveL 5917 to (502.8, 490.4, 12.8) mm, rotated rx 0 ry 90 rz 0 deg; joints [-11.076, -27.625, 111.311, -15.087, -83.04, 50.868]
  Call Extruder(0.198)
  MoveL 5918 to (509.6, 490.4, 12.8) mm, rotated rx 0 ry 90 rz 0 deg; joints [-10.955, -27.494, 110.494, -14.988, -82.373, 51.034]
  Call Extruder(0.170)
  MoveL 5919 to (509.6, 496.25, 12.8) mm, rotated rx 0 ry 90 rz 0 deg; joints [-11.486, -27.471, 110.354, -15.527, -82.278, 51.129]
  Call Extruder(0.056)
  MoveL 5920 to (507.67, 496.26, 12.8) mm, rotated rx 0 ry 90 rz 0 deg; joints [-11.521, -27.509, 110.587, -15.556, -82.466, 51.081]
  Call Extruder(0.073)
  MoveL 5921 to (507.67, 498.75, 12.8) mm, rotated rx 0 ry 90 rz 0 deg; joints [-11.748, -27.499, 110.525, -15.786, -82.424, 51.121]
  Call Extruder(0.056)
  MoveL 5922 to (509.6, 498.75, 12.8) mm, rotated rx 0 ry 90 rz 0 deg; joints [-11.712, -27.461, 110.292, -15.757, -82.235, 51.17]
  Call Extruder(0.037)
  MoveL 5923 to (509.6, 500.01, 12.8) mm, rotated rx 0 ry 90 rz 0 deg; joints [-11.825, -27.456, 110.261, -15.872, -82.214, 51.191]
  Call Extruder(0.010)
  MoveL 5924 to (509.6, 500.36, 12.8) mm, rotated rx 0 ry 90 rz 0 deg; joints [-11.857, -27.454, 110.252, -15.905, -82.208, 51.197]
  Call Extruder(0.007)
  MoveL 5925 to (509.25, 500.36, 12.8) mm, rotated rx 0 ry 90 rz 0 deg; joints [-11.863, -27.461, 110.294, -15.91, -82.242, 51.188]
  Call Extruder(0.036)
  MoveL 5926 to (508.02, 500.36, 12.8) mm, rotated rx 0 ry 90 rz 0 deg; joints [-11.886, -27.486, 110.442, -15.929, -82.362, 51.157]
  Call Extruder(0.010)
  MoveL 5927 to (507.67, 500.36, 12.8) mm, rotated rx 0 ry 90 rz 0 deg; joints [-11.893, -27.493, 110.484, -15.934, -82.396, 51.148]
  Call Extruder(0.007)
  MoveL 5928 to (507.67, 500.71, 12.8) mm, rotated rx 0 ry 90 rz 0 deg; joints [-11.925, -27.491, 110.476, -15.966, -82.39, 51.154]
  Call Extruder(0.062)
  MoveL 5929 to (507.67, 502.84, 12.8) mm, rotated rx 0 ry 90 rz 0 deg; joints [-12.118, -27.482, 110.421, -16.163, -82.353, 51.189]
  Call Extruder(0.056)
  MoveL 5930 to (509.6, 502.85, 12.8) mm, rotated rx 0 ry 90 rz 0 deg; joints [-12.081, -27.444, 110.188, -16.133, -82.165, 51.239]
  Call Extruder(0.197)
  MoveL 5931 to (509.6, 509.6, 12.8) mm, rotated rx 0 ry 90 rz 0 deg; joints [-12.688, -27.414, 110.01, -16.751, -82.044, 51.357]
  Call Extruder(0.559)
  MoveL 5932 to (490.4, 509.6, 12.8) mm, rotated rx 0 ry 90 rz 0 deg; joints [-13.088, -27.773, 112.297, -17.085, -83.902, 50.835]
  MoveL 5933 to (490.4, 490.4, 12.8) mm, rotated rx 0 ry 90 rz 0 deg; joints [-11.303, -27.843, 112.787, -15.279, -84.26, 50.559]
  Call Extruder(0.183)
  MoveL 5934 to (496.68, 490.4, 12.8) mm, rotated rx 0 ry 90 rz 0 deg; joints [-11.187, -27.736, 112.043, -15.18, -83.642, 50.717]
  Call Extruder(0.055)
  MoveL 5935 to (496.68, 492.3, 12.8) mm, rotated rx 0 ry 90 rz 0 deg; joints [-11.363, -27.729, 111.998, -15.358, -83.61, 50.744]
  Call Extruder(0.072)
  MoveL 5936 to (499.13, 492.3, 12.8) mm, rotated rx 0 ry 90 rz 0 deg; joints [-11.317, -27.685, 111.705, -15.319, -83.368, 50.806]
  Call Extruder(0.055)
  MoveL 5937 to (499.14, 490.4, 12.8) mm, rotated rx 0 ry 90 rz 0 deg; joints [-11.142, -27.692, 111.75, -15.142, -83.4, 50.778]
  Call Extruder(0.026)
  MoveL 5938 to (500.03, 490.4, 12.8) mm, rotated rx 0 ry 90 rz 0 deg; joints [-11.126, -27.676, 111.643, -15.128, -83.313, 50.8]
  Call Extruder(0.055)
  MoveL 5939 to (500.03, 492.3, 12.8) mm, rotated rx 0 ry 90 rz 0 deg; joints [-11.301, -27.669, 111.598, -15.306, -83.281, 50.828]
  Call Extruder(0.060)
  MoveL 5940 to (502.1, 492.3, 12.8) mm, rotated rx 0 ry 90 rz 0 deg; joints [-11.263, -27.631, 111.35, -15.274, -83.077, 50.88]
  Call Extruder(0.007)
  MoveL 5941 to (502.45, 492.3, 12.8) mm, rotated rx 0 ry 90 rz 0 deg; joints [-11.256, -27.624, 111.308, -15.269, -83.043, 50.888]
  Set speed (120.0 mm/s)
  MoveL 5942 to (502.45, 491.95, 12.8) mm, rotated rx 0 ry 90 rz 0 deg; joints [-11.224, -27.626, 111.317, -15.236, -83.049, 50.883]
  Set speed (1000.0 mm/s)
  MoveL 5943 to (502.45, 491.9, 12.8) mm, rotated rx 0 ry 90 rz 0 deg; joints [-11.22, -27.626, 111.318, -15.231, -83.05, 50.882]
  Set speed (1000.0 mm/s)
  MoveL 5944 to (502.55, 491.9, 12.8) mm, rotated rx 0 ry 90 rz 0 deg; joints [-11.218, -27.624, 111.306, -15.23, -83.04, 50.885]
  Set speed (1000.0 mm/s)
  MoveL 5945 to (500, 492.33, 12.8) mm, rotated rx 0 ry 90 rz 0 deg; joints [-11.304, -27.669, 111.601, -15.309, -83.283, 50.828]
  Set speed (1000.0 mm/s)
  MoveL 5946 to (499.58, 491.85, 12.8) mm, rotated rx 0 ry 90 rz 0 deg; joints [-11.268, -27.679, 111.662, -15.271, -83.332, 50.81]
  Set speed (15.0 mm/s)
  Call Extruder(0.005)
  MoveL 5947 to (499.58, 492.35, 12.8) mm, rotated rx 0 ry 90 rz 0 deg; joints [-11.313, -27.677, 111.651, -15.317, -83.324, 50.817]
  Call Extruder(0.015)
  MoveL 5948 to (499.58, 490.86, 12.8) mm, rotated rx 0 ry 90 rz 0 deg; joints [-11.176, -27.682, 111.686, -15.178, -83.349, 50.796]
  Set speed (120.0 mm/s)
  MoveL 5949 to (499.84, 490.75, 12.8) mm, rotated rx 0 ry 90 rz 0 deg; joints [-11.161, -27.678, 111.658, -15.164, -83.326, 50.8]
  Set speed (1000.0 mm/s)
  MoveL 5950 to (499.16, 492.33, 12.8) mm, rotated rx 0 ry 90 rz 0 deg; joints [-11.319, -27.685, 111.701, -15.322, -83.365, 50.807]
  Set speed (1000.0 mm/s)
  MoveL 5951 to (496.65, 492.33, 12.8) mm, rotated rx 0 ry 90 rz 0 deg; joints [-11.366, -27.73, 112, -15.361, -83.612, 50.743]
  Set speed (1000.0 mm/s)
  MoveL 5952 to (490.68, 490.68, 12.8) mm, rotated rx 0 ry 90 rz 0 deg; joints [-11.324, -27.837, 112.748, -15.301, -84.228, 50.57]
  Set speed (1000.0 mm/s)
  MoveL 5953 to (490.68, 490.68, 12.9) mm, rotated rx 0 ry 90 rz 0 deg; joints [-11.324, -27.848, 112.753, -15.301, -84.222, 50.571]
  Set speed (30.0 mm/s)
  Call Extruder(0.767)
  MoveL 5954 to (509.32, 509.32, 12.9) mm, rotated rx 0 ry 90 rz 0 deg; joints [-12.669, -27.431, 110.056, -16.73, -82.072, 51.346]
  MoveL 5955 to (509.44, 509.44, 12.9) mm, rotated rx 0 ry 90 rz 0 deg; joints [-12.677, -27.428, 110.038, -16.74, -82.057, 51.351]
  Set speed (120.0 mm/s)
  MoveL 5956 to (507.39, 502.51, 12.9) mm, rotated rx 0 ry 90 rz 0 deg; joints [-12.094, -27.5, 110.468, -16.137, -82.381, 51.178]
  Set speed (30.0 mm/s)
  Call Extruder(0.280)
  MoveL 5957 to (500.58, 509.32, 12.9) mm, rotated rx 0 ry 90 rz 0 deg; joints [-12.847, -27.602, 111.103, -16.877, -82.916, 51.111]
  Set speed (120.0 mm/s)
  MoveL 5958 to (499.42, 509.32, 12.9) mm, rotated rx 0 ry 90 rz 0 deg; joints [-12.872, -27.624, 111.241, -16.897, -83.029, 51.08]
  Set speed (30.0 mm/s)
  Call Extruder(0.360)
  MoveL 5959 to (490.68, 500.58, 12.9) mm, rotated rx 0 ry 90 rz 0 deg; joints [-12.247, -27.813, 112.509, -16.234, -84.043, 50.709]
  Set speed (120.0 mm/s)
  MoveL 5960 to (490.68, 499.42, 12.9) mm, rotated rx 0 ry 90 rz 0 deg; joints [-12.139, -27.818, 112.538, -16.125, -84.065, 50.692]
  Set speed (30.0 mm/s)
  Call Extruder(0.282)
  MoveL 5961 to (497.52, 492.58, 12.9) mm, rotated rx 0 ry 90 rz 0 deg; joints [-11.373, -27.724, 111.896, -15.371, -83.517, 50.77]
  MoveL 5962 to (497.64, 492.46, 12.9) mm, rotated rx 0 ry 90 rz 0 deg; joints [-11.359, -27.722, 111.884, -15.357, -83.507, 50.772]
  Set speed (120.0 mm/s)
  MoveL 5963 to (502.48, 492.58, 12.9) mm, rotated rx 0 ry 90 rz 0 deg; joints [-11.281, -27.633, 111.304, -15.294, -83.03, 50.895]
  Set speed (30.0 mm/s)
  Call Extruder(0.202)
  MoveL 5964 to (507.39, 497.49, 12.9) mm, rotated rx 0 ry 90 rz 0 deg; joints [-11.639, -27.52, 110.595, -15.674, -82.467, 51.095]
  MoveL 5965 to (507.51, 497.61, 12.9) mm, rotated rx 0 ry 90 rz 0 deg; joints [-11.647, -27.517, 110.577, -15.684, -82.453, 51.1]
  Set speed (120.0 mm/s)
  MoveL 5966 to (508.87, 498.97, 12.9) mm, rotated rx 0 ry 90 rz 0 deg; joints [-11.745, -27.485, 110.379, -15.789, -82.297, 51.157]
  Set speed (30.0 mm/s)
  Call Extruder(0.018)
  MoveL 5967 to (509.32, 499.42, 12.9) mm, rotated rx 0 ry 90 rz 0 deg; joints [-11.777, -27.474, 110.314, -15.823, -82.246, 51.176]
  Set speed (120.0 mm/s)
  MoveL 5968 to (507.64, 498.72, 12.9) mm, rotated rx 0 ry 90 rz 0 deg; joints [-11.746, -27.51, 110.534, -15.784, -82.422, 51.122]
  Set speed (1000.0 mm/s)
  MoveL 5969 to (507.64, 496.17, 12.9) mm, rotated rx 0 ry 90 rz 0 deg; joints [-11.514, -27.521, 110.597, -15.549, -82.465, 51.08]
  Set speed (1000.0 mm/s)
  MoveL 5970 to (509.32, 490.68, 12.9) mm, rotated rx 0 ry 90 rz 0 deg; joints [-10.985, -27.509, 110.527, -15.018, -82.391, 51.033]
  Set speed (30.0 mm/s)
  Call Extruder(0.767)
  MoveL 5971 to (490.68, 509.32, 12.9) mm, rotated rx 0 ry 90 rz 0 deg; joints [-13.056, -27.78, 112.277, -17.053, -83.875, 50.84]
  MoveL 5972 to (490.56, 509.44, 12.9) mm, rotated rx 0 ry 90 rz 0 deg; joints [-13.07, -27.782, 112.288, -17.067, -83.885, 50.838]
  Set speed (120.0 mm/s)
  MoveL 5973 to (502.59, 492.37, 12.9) mm, rotated rx 0 ry 90 rz 0 deg; joints [-11.26, -27.632, 111.296, -15.273, -83.023, 50.894]
  Set speed (1000.0 mm/s)
  MoveL 5974 to (502.52, 492.3, 12.9) mm, rotated rx 0 ry 90 rz 0 deg; joints [-11.255, -27.634, 111.306, -15.268, -83.031, 50.891]
  Set speed (15.0 mm/s)
  Call Extruder(0.010)
  MoveL 5975 to (502.52, 491.95, 12.9) mm, rotated rx 0 ry 90 rz 0 deg; joints [-11.223, -27.635, 111.314, -15.235, -83.037, 50.886]
  Call Extruder(0.035)
  MoveL 5976 to (502.51, 490.75, 12.9) mm, rotated rx 0 ry 90 rz 0 deg; joints [-11.113, -27.639, 111.343, -15.124, -83.057, 50.868]
  Call Extruder(0.010)
  MoveL 5977 to (502.52, 490.4, 12.9) mm, rotated rx 0 ry 90 rz 0 deg; joints [-11.081, -27.641, 111.351, -15.091, -83.063, 50.863]
  Call Extruder(0.007)
  MoveL 5978 to (502.87, 490.4, 12.9) mm, rotated rx 0 ry 90 rz 0 deg; joints [-11.075, -27.634, 111.309, -15.086, -83.029, 50.871]
  Call Extruder(0.196)
  MoveL 5979 to (509.6, 490.4, 12.9) mm, rotated rx 0 ry 90 rz 0 deg; joints [-10.955, -27.505, 110.499, -14.988, -82.368, 51.036]
  Call Extruder(0.169)
  MoveL 5980 to (509.6, 496.19, 12.9) mm, rotated rx 0 ry 90 rz 0 deg; joints [-11.48, -27.482, 110.361, -15.522, -82.273, 51.129]
  Call Extruder(0.056)
  MoveL 5981 to (507.67, 496.2, 12.9) mm, rotated rx 0 ry 90 rz 0 deg; joints [-11.516, -27.52, 110.593, -15.551, -82.462, 51.081]
  Call Extruder(0.063)
  MoveL 5982 to (507.67, 498.35, 12.9) mm, rotated rx 0 ry 90 rz 0 deg; joints [-11.711, -27.511, 110.54, -15.749, -82.425, 51.116]
  Call Extruder(0.010)
  MoveL 5983 to (507.67, 498.7, 12.9) mm, rotated rx 0 ry 90 rz 0 deg; joints [-11.743, -27.51, 110.531, -15.781, -82.419, 51.122]
  Call Extruder(0.007)
  MoveL 5984 to (508.02, 498.7, 12.9) mm, rotated rx 0 ry 90 rz 0 deg; joints [-11.736, -27.503, 110.489, -15.776, -82.385, 51.131]
  Call Extruder(0.046)
  MoveL 5985 to (509.6, 498.69, 12.9) mm, rotated rx 0 ry 90 rz 0 deg; joints [-11.706, -27.472, 110.299, -15.752, -82.231, 51.171]
  Call Extruder(0.050)
  MoveL 5986 to (509.6, 500.42, 12.9) mm, rotated rx 0 ry 90 rz 0 deg; joints [-11.862, -27.464, 110.255, -15.91, -82.202, 51.2]
  Call Extruder(0.046)
  MoveL 5987 to (508.02, 500.41, 12.9) mm, rotated rx 0 ry 90 rz 0 deg; joints [-11.892, -27.496, 110.446, -15.934, -82.356, 51.159]
  Call Extruder(0.010)
  MoveL 5988 to (507.67, 500.41, 12.9) mm, rotated rx 0 ry 90 rz 0 deg; joints [-11.898, -27.503, 110.488, -15.94, -82.39, 51.15]
  Call Extruder(0.007)
  MoveL 5989 to (507.67, 500.76, 12.9) mm, rotated rx 0 ry 90 rz 0 deg; joints [-11.93, -27.501, 110.479, -15.972, -82.384, 51.156]
  Call Extruder(0.062)
  MoveL 5990 to (507.67, 502.9, 12.9) mm, rotated rx 0 ry 90 rz 0 deg; joints [-12.123, -27.492, 110.425, -16.168, -82.347, 51.192]
  Call Extruder(0.056)
  MoveL 5991 to (509.6, 502.9, 12.9) mm, rotated rx 0 ry 90 rz 0 deg; joints [-12.086, -27.454, 110.192, -16.138, -82.159, 51.242]
  Call Extruder(0.195)
  MoveL 5992 to (509.6, 509.6, 12.9) mm, rotated rx 0 ry 90 rz 0 deg; joints [-12.688, -27.424, 110.015, -16.751, -82.039, 51.358]
  Call Extruder(0.559)
  MoveL 5993 to (490.4, 509.6, 12.9) mm, rotated rx 0 ry 90 rz 0 deg; joints [-13.088, -27.784, 112.302, -17.085, -83.897, 50.836]
  MoveL 5994 to (490.4, 490.4, 12.9) mm, rotated rx 0 ry 90 rz 0 deg; joints [-11.303, -27.853, 112.792, -15.279, -84.255, 50.56]
  Call Extruder(0.171)
  MoveL 5995 to (496.27, 490.4, 12.9) mm, rotated rx 0 ry 90 rz 0 deg; joints [-11.194, -27.754, 112.096, -15.186, -83.677, 50.708]
  Call Extruder(0.010)
  MoveL 5996 to (496.62, 490.4, 12.9) mm, rotated rx 0 ry 90 rz 0 deg; joints [-11.188, -27.747, 112.055, -15.181, -83.642, 50.717]
  Call Extruder(0.007)
  MoveL 5997 to (496.62, 490.75, 12.9) mm, rotated rx 0 ry 90 rz 0 deg; joints [-11.22, -27.746, 112.046, -15.214, -83.636, 50.722]
  Call Extruder(0.035)
  MoveL 5998 to (496.62, 491.95, 12.9) mm, rotated rx 0 ry 90 rz 0 deg; joints [-11.331, -27.742, 112.018, -15.326, -83.616, 50.739]
  Call Extruder(0.010)
  MoveL 5999 to (496.62, 492.3, 12.9) mm, rotated rx 0 ry 90 rz 0 deg; joints [-11.364, -27.741, 112.01, -15.359, -83.61, 50.744]
  Call Extruder(0.007)
  MoveL 6000 to (496.97, 492.3, 12.9) mm, rotated rx 0 ry 90 rz 0 deg; joints [-11.357, -27.735, 111.968, -15.353, -83.576, 50.753]
  Call Extruder(0.061)
  MoveL 6001 to (499.08, 492.3, 12.9) mm, rotated rx 0 ry 90 rz 0 deg; joints [-11.318, -27.697, 111.717, -15.321, -83.369, 50.806]
  Call Extruder(0.055)
  MoveL 6002 to (499.08, 490.4, 12.9) mm, rotated rx 0 ry 90 rz 0 deg; joints [-11.143, -27.704, 111.762, -15.143, -83.401, 50.778]
  Call Extruder(0.029)
  MoveL 6003 to (500.09, 490.4, 12.9) mm, rotated rx 0 ry 90 rz 0 deg; joints [-11.125, -27.685, 111.641, -15.128, -83.301, 50.803]
  Call Extruder(0.055)
  MoveL 6004 to (500.09, 492.3, 12.9) mm, rotated rx 0 ry 90 rz 0 deg; joints [-11.3, -27.678, 111.596, -15.305, -83.269, 50.831]
  Call Extruder(0.060)
  MoveL 6005 to (502.17, 492.3, 12.9) mm, rotated rx 0 ry 90 rz 0 deg; joints [-11.262, -27.64, 111.348, -15.273, -83.066, 50.883]
  Call Extruder(0.007)
  MoveL 6006 to (502.52, 492.3, 12.9) mm, rotated rx 0 ry 90 rz 0 deg; joints [-11.255, -27.634, 111.306, -15.268, -83.031, 50.891]
  Set speed (120.0 mm/s)
  MoveL 6007 to (502.52, 491.95, 12.9) mm, rotated rx 0 ry 90 rz 0 deg; joints [-11.223, -27.635, 111.314, -15.235, -83.037, 50.886]
  Set speed (1000.0 mm/s)
  MoveL 6008 to (502.52, 491.9, 12.9) mm, rotated rx 0 ry 90 rz 0 deg; joints [-11.218, -27.635, 111.315, -15.231, -83.038, 50.885]
  Set speed (1000.0 mm/s)
  MoveL 6009 to (502.62, 491.9, 12.9) mm, rotated rx 0 ry 90 rz 0 deg; joints [-11.217, -27.633, 111.303, -15.229, -83.028, 50.888]
  Set speed (1000.0 mm/s)
  MoveL 6010 to (500.07, 492.33, 12.9) mm, rotated rx 0 ry 90 rz 0 deg; joints [-11.303, -27.679, 111.598, -15.308, -83.271, 50.831]
  Set speed (1000.0 mm/s)
  MoveL 6011 to (499.58, 491.66, 12.9) mm, rotated rx 0 ry 90 rz 0 deg; joints [-11.25, -27.69, 111.672, -15.253, -83.33, 50.809]
  Set speed (15.0 mm/s)
  Call Extruder(0.006)
  MoveL 6012 to (499.58, 491.17, 12.9) mm, rotated rx 0 ry 90 rz 0 deg; joints [-11.205, -27.692, 111.683, -15.207, -83.338, 50.802]
  Call Extruder(0.005)
  MoveL 6013 to (499.7, 490.79, 12.9) mm, rotated rx 0 ry 90 rz 0 deg; joints [-11.168, -27.691, 111.678, -15.17, -83.333, 50.799]
  Call Extruder(0.021)
  MoveL 6014 to (499.51, 492.58, 12.9) mm, rotated rx 0 ry 90 rz 0 deg; joints [-11.336, -27.688, 111.658, -15.34, -83.321, 50.821]
  Set speed (120.0 mm/s)
  MoveL 6015 to (499.57, 492.8, 12.9) mm, rotated rx 0 ry 90 rz 0 deg; joints [-11.355, -27.686, 111.646, -15.359, -83.312, 50.825]
  Set speed (1000.0 mm/s)
  MoveL 6016 to (496.89, 492.38, 12.9) mm, rotated rx 0 ry 90 rz 0 deg; joints [-11.366, -27.736, 111.976, -15.362, -83.582, 50.752]
  Set speed (1000.0 mm/s)
  MoveL 6017 to (490.68, 490.68, 12.9) mm, rotated rx 0 ry 90 rz 0 deg; joints [-11.324, -27.848, 112.753, -15.301, -84.222, 50.571]
  Set speed (1000.0 mm/s)
  MoveL 6018 to (490.68, 490.68, 13) mm, rotated rx 0 ry 90 rz 0 deg; joints [-11.324, -27.859, 112.758, -15.301, -84.217, 50.572]
  Set speed (30.0 mm/s)
  Call Extruder(0.767)
  MoveL 6019 to (509.32, 509.32, 13) mm, rotated rx 0 ry 90 rz 0 deg; joints [-12.669, -27.441, 110.061, -16.731, -82.066, 51.347]
  MoveL 6020 to (509.44, 509.44, 13) mm, rotated rx 0 ry 90 rz 0 deg; joints [-12.677, -27.438, 110.043, -16.74, -82.052, 51.353]
  Set speed (120.0 mm/s)
  MoveL 6021 to (507.39, 502.51, 13) mm, rotated rx 0 ry 90 rz 0 deg; joints [-12.094, -27.51, 110.474, -16.137, -82.376, 51.179]
  Set speed (30.0 mm/s)
  Call Extruder(0.280)
  MoveL 6022 to (500.58, 509.32, 13) mm, rotated rx 0 ry 90 rz 0 deg; joints [-12.847, -27.613, 111.108, -16.877, -82.911, 51.113]
  Set speed (120.0 mm/s)
  MoveL 6023 to (499.42, 509.32, 13) mm, rotated rx 0 ry 90 rz 0 deg; joints [-12.872, -27.634, 111.247, -16.897, -83.023, 51.081]
  Set speed (30.0 mm/s)
  Call Extruder(0.360)
  MoveL 6024 to (490.68, 500.58, 13) mm, rotated rx 0 ry 90 rz 0 deg; joints [-12.247, -27.824, 112.514, -16.234, -84.038, 50.711]
  Set speed (120.0 mm/s)
  MoveL 6025 to (490.68, 499.42, 13) mm, rotated rx 0 ry 90 rz 0 deg; joints [-12.139, -27.828, 112.544, -16.125, -84.06, 50.694]
  Set speed (30.0 mm/s)
  Call Extruder(0.282)
  MoveL 6026 to (497.52, 492.58, 13) mm, rotated rx 0 ry 90 rz 0 deg; joints [-11.373, -27.734, 111.901, -15.371, -83.512, 50.772]
  MoveL 6027 to (497.64, 492.46, 13) mm, rotated rx 0 ry 90 rz 0 deg; joints [-11.359, -27.733, 111.889, -15.358, -83.502, 50.773]
  Set speed (120.0 mm/s)
  MoveL 6028 to (502.48, 492.58, 13) mm, rotated rx 0 ry 90 rz 0 deg; joints [-11.281, -27.644, 111.309, -15.295, -83.025, 50.896]
  Set speed (30.0 mm/s)
  Call Extruder(0.202)
  MoveL 6029 to (507.39, 497.49, 13) mm, rotated rx 0 ry 90 rz 0 deg; joints [-11.639, -27.531, 110.6, -15.675, -82.462, 51.096]
  MoveL 6030 to (507.51, 497.61, 13) mm, rotated rx 0 ry 90 rz 0 deg; joints [-11.647, -27.528, 110.582, -15.684, -82.448, 51.102]
  Set speed (120.0 mm/s)
  MoveL 6031 to (508.82, 498.92, 13) mm, rotated rx 0 ry 90 rz 0 deg; joints [-11.741, -27.497, 110.393, -15.784, -82.299, 51.156]
  Set speed (30.0 mm/s)
  Call Extruder(0.021)
  MoveL 6032 to (509.32, 499.42, 13) mm, rotated rx 0 ry 90 rz 0 deg; joints [-11.777, -27.485, 110.32, -15.823, -82.241, 51.177]
  Set speed (120.0 mm/s)
  MoveL 6033 to (507.64, 498.67, 13) mm, rotated rx 0 ry 90 rz 0 deg; joints [-11.74, -27.521, 110.54, -15.779, -82.417, 51.122]
  Set speed (1000.0 mm/s)
  MoveL 6034 to (507.64, 496.11, 13) mm, rotated rx 0 ry 90 rz 0 deg; joints [-11.509, -27.531, 110.604, -15.543, -82.461, 51.08]
  Set speed (1000.0 mm/s)
  MoveL 6035 to (509.32, 490.68, 13) mm, rotated rx 0 ry 90 rz 0 deg; joints [-10.985, -27.52, 110.532, -15.018, -82.386, 51.035]
  Set speed (30.0 mm/s)
  Call Extruder(0.767)
  MoveL 6036 to (490.68, 509.32, 13) mm, rotated rx 0 ry 90 rz 0 deg; joints [-13.056, -27.791, 112.282, -17.054, -83.87, 50.841]
  MoveL 6037 to (490.56, 509.44, 13) mm, rotated rx 0 ry 90 rz 0 deg; joints [-13.07, -27.792, 112.293, -17.067, -83.88, 50.84]
  Set speed (120.0 mm/s)
  MoveL 6038 to (502.65, 492.37, 13) mm, rotated rx 0 ry 90 rz 0 deg; joints [-11.259, -27.642, 111.293, -15.273, -83.012, 50.897]
  Set speed (1000.0 mm/s)
  MoveL 6039 to (502.58, 492.3, 13) mm, rotated rx 0 ry 90 rz 0 deg; joints [-11.254, -27.643, 111.303, -15.267, -83.02, 50.894]
  Set speed (15.0 mm/s)
  Call Extruder(0.010)
  MoveL 6040 to (502.58, 491.95, 13) mm, rotated rx 0 ry 90 rz 0 deg; joints [-11.222, -27.644, 111.312, -15.235, -83.026, 50.889]
  Call Extruder(0.035)
  MoveL 6041 to (502.58, 490.75, 13) mm, rotated rx 0 ry 90 rz 0 deg; joints [-11.112, -27.649, 111.34, -15.123, -83.046, 50.871]
  Call Extruder(0.010)
  MoveL 6042 to (502.58, 490.4, 13) mm, rotated rx 0 ry 90 rz 0 deg; joints [-11.08, -27.65, 111.348, -15.09, -83.052, 50.866]
  Call Extruder(0.007)
  MoveL 6043 to (502.93, 490.4, 13) mm, rotated rx 0 ry 90 rz 0 deg; joints [-11.073, -27.644, 111.306, -15.085, -83.017, 50.874]
  Call Extruder(0.194)
  MoveL 6044 to (509.6, 490.4, 13) mm, rotated rx 0 ry 90 rz 0 deg; joints [-10.955, -27.515, 110.504, -14.988, -82.363, 51.037]
  Call Extruder(0.167)
  MoveL 6045 to (509.6, 496.13, 13) mm, rotated rx 0 ry 90 rz 0 deg; joints [-11.475, -27.493, 110.367, -15.517, -82.269, 51.13]
  Call Extruder(0.056)
  MoveL 6046 to (507.67, 496.14, 13) mm, rotated rx 0 ry 90 rz 0 deg; joints [-11.511, -27.531, 110.6, -15.546, -82.458, 51.082]
  Call Extruder(0.063)
  MoveL 6047 to (507.67, 498.29, 13) mm, rotated rx 0 ry 90 rz 0 deg; joints [-11.706, -27.522, 110.546, -15.744, -82.421, 51.117]
  Call Extruder(0.010)
  MoveL 6048 to (507.67, 498.64, 13) mm, rotated rx 0 ry 90 rz 0 deg; joints [-11.737, -27.521, 110.538, -15.776, -82.415, 51.122]
  Call Extruder(0.007)
  MoveL 6049 to (508.02, 498.64, 13) mm, rotated rx 0 ry 90 rz 0 deg; joints [-11.731, -27.514, 110.496, -15.771, -82.381, 51.131]
  Call Extruder(0.046)
  MoveL 6050 to (509.6, 498.64, 13) mm, rotated rx 0 ry 90 rz 0 deg; joints [-11.701, -27.482, 110.305, -15.747, -82.227, 51.171]
  Call Extruder(0.043)
  MoveL 6051 to (509.6, 500.12, 13) mm, rotated rx 0 ry 90 rz 0 deg; joints [-11.835, -27.476, 110.268, -15.883, -82.202, 51.196]
  Call Extruder(0.010)
  MoveL 6052 to (509.6, 500.47, 13) mm, rotated rx 0 ry 90 rz 0 deg; joints [-11.867, -27.475, 110.259, -15.915, -82.196, 51.202]
  Call Extruder(0.007)
  MoveL 6053 to (509.25, 500.47, 13) mm, rotated rx 0 ry 90 rz 0 deg; joints [-11.873, -27.482, 110.301, -15.921, -82.23, 51.193]
  Call Extruder(0.036)
  MoveL 6054 to (508.02, 500.47, 13) mm, rotated rx 0 ry 90 rz 0 deg; joints [-11.897, -27.506, 110.45, -15.939, -82.35, 51.162]
  Call Extruder(0.010)
  MoveL 6055 to (507.67, 500.47, 13) mm, rotated rx 0 ry 90 rz 0 deg; joints [-11.903, -27.513, 110.492, -15.945, -82.384, 51.153]
  Call Extruder(0.007)
  MoveL 6056 to (507.67, 500.82, 13) mm, rotated rx 0 ry 90 rz 0 deg; joints [-11.935, -27.512, 110.483, -15.977, -82.378, 51.158]
  Call Extruder(0.062)
  MoveL 6057 to (507.67, 502.96, 13) mm, rotated rx 0 ry 90 rz 0 deg; joints [-12.128, -27.503, 110.428, -16.174, -82.34, 51.194]
  Call Extruder(0.056)
  MoveL 6058 to (509.6, 502.96, 13) mm, rotated rx 0 ry 90 rz 0 deg; joints [-12.091, -27.464, 110.196, -16.144, -82.153, 51.244]
  Call Extruder(0.193)
  MoveL 6059 to (509.6, 509.6, 13) mm, rotated rx 0 ry 90 rz 0 deg; joints [-12.688, -27.434, 110.02, -16.752, -82.034, 51.36]
  Call Extruder(0.559)
  MoveL 6060 to (490.4, 509.6, 13) mm, rotated rx 0 ry 90 rz 0 deg; joints [-13.088, -27.794, 112.308, -17.085, -83.892, 50.838]
  MoveL 6061 to (490.4, 490.4, 13) mm, rotated rx 0 ry 90 rz 0 deg; joints [-11.303, -27.864, 112.798, -15.279, -84.25, 50.562]
  Call Extruder(0.169)
  MoveL 6062 to (496.21, 490.4, 13) mm, rotated rx 0 ry 90 rz 0 deg; joints [-11.195, -27.765, 112.108, -15.187, -83.677, 50.708]
  Call Extruder(0.010)
  MoveL 6063 to (496.56, 490.4, 13) mm, rotated rx 0 ry 90 rz 0 deg; joints [-11.189, -27.759, 112.067, -15.182, -83.643, 50.717]
  Call Extruder(0.007)
  MoveL 6064 to (496.56, 490.75, 13) mm, rotated rx 0 ry 90 rz 0 deg; joints [-11.221, -27.758, 112.058, -15.215, -83.637, 50.722]
  Call Extruder(0.035)
  MoveL 6065 to (496.56, 491.95, 13) mm, rotated rx 0 ry 90 rz 0 deg; joints [-11.333, -27.754, 112.03, -15.327, -83.616, 50.739]
  Call Extruder(0.010)
  MoveL 6066 to (496.56, 492.3, 13) mm, rotated rx 0 ry 90 rz 0 deg; joints [-11.365, -27.752, 112.022, -15.36, -83.61, 50.744]
  Call Extruder(0.007)
  MoveL 6067 to (496.91, 492.3, 13) mm, rotated rx 0 ry 90 rz 0 deg; joints [-11.358, -27.746, 111.98, -15.354, -83.576, 50.753]
  Call Extruder(0.061)
  MoveL 6068 to (499.02, 492.3, 13) mm, rotated rx 0 ry 90 rz 0 deg; joints [-11.319, -27.708, 111.729, -15.322, -83.369, 50.806]
  Call Extruder(0.055)
  MoveL 6069 to (499.02, 490.4, 13) mm, rotated rx 0 ry 90 rz 0 deg; joints [-11.144, -27.715, 111.773, -15.144, -83.401, 50.778]
  Call Extruder(0.033)
  MoveL 6070 to (500.15, 490.4, 13) mm, rotated rx 0 ry 90 rz 0 deg; joints [-11.123, -27.695, 111.638, -15.127, -83.29, 50.806]
  Call Extruder(0.055)
  MoveL 6071 to (500.16, 492.3, 13) mm, rotated rx 0 ry 90 rz 0 deg; joints [-11.298, -27.688, 111.593, -15.304, -83.258, 50.834]
  Call Extruder(0.060)
  MoveL 6072 to (502.23, 492.3, 13) mm, rotated rx 0 ry 90 rz 0 deg; joints [-11.26, -27.65, 111.345, -15.272, -83.054, 50.886]
  Call Extruder(0.007)
  MoveL 6073 to (502.58, 492.3, 13) mm, rotated rx 0 ry 90 rz 0 deg; joints [-11.254, -27.643, 111.303, -15.267, -83.02, 50.894]
  Set speed (120.0 mm/s)
  MoveL 6074 to (502.58, 491.95, 13) mm, rotated rx 0 ry 90 rz 0 deg; joints [-11.222, -27.644, 111.312, -15.235, -83.026, 50.889]
  Set speed (1000.0 mm/s)
  MoveL 6075 to (502.58, 491.9, 13) mm, rotated rx 0 ry 90 rz 0 deg; joints [-11.217, -27.645, 111.313, -15.23, -83.027, 50.888]
  Set speed (1000.0 mm/s)
  MoveL 6076 to (502.68, 491.9, 13) mm, rotated rx 0 ry 90 rz 0 deg; joints [-11.215, -27.643, 111.301, -15.228, -83.017, 50.891]
  Set speed (1000.0 mm/s)
  MoveL 6077 to (500.13, 492.33, 13) mm, rotated rx 0 ry 90 rz 0 deg; joints [-11.302, -27.688, 111.596, -15.307, -83.26, 50.834]
  Set speed (1000.0 mm/s)
  MoveL 6078 to (499.59, 492.34, 13) mm, rotated rx 0 ry 90 rz 0 deg; joints [-11.313, -27.698, 111.66, -15.317, -83.313, 50.82]
  Set speed (15.0 mm/s)
  Call Extruder(0.007)
  MoveL 6079 to (499.78, 492.64, 13) mm, rotated rx 0 ry 90 rz 0 deg; joints [-11.337, -27.693, 111.63, -15.342, -83.289, 50.83]
  Call Extruder(0.034)
  MoveL 6080 to (499.53, 490.91, 13) mm, rotated rx 0 ry 90 rz 0 deg; joints [-11.182, -27.704, 111.701, -15.184, -83.342, 50.798]
  Set speed (120.0 mm/s)
  MoveL 6081 to (499.45, 491.09, 13) mm, rotated rx 0 ry 90 rz 0 deg; joints [-11.2, -27.705, 111.706, -15.202, -83.347, 50.799]
  Set speed (1000.0 mm/s)
  MoveL 6082 to (496.53, 492.33, 13) mm, rotated rx 0 ry 90 rz 0 deg; joints [-11.368, -27.753, 112.024, -15.363, -83.613, 50.744]
  Set speed (1000.0 mm/s)
  MoveL 6083 to (490.68, 490.68, 13) mm, rotated rx 0 ry 90 rz 0 deg; joints [-11.324, -27.859, 112.758, -15.301, -84.217, 50.572]
  Set speed (1000.0 mm/s)
  MoveL 6084 to (490.68, 490.68, 13.1) mm, rotated rx 0 ry 90 rz 0 deg; joints [-11.324, -27.869, 112.763, -15.301, -84.212, 50.574]
  Set speed (30.0 mm/s)
  Call Extruder(0.767)
  MoveL 6085 to (509.32, 509.32, 13.1) mm, rotated rx 0 ry 90 rz 0 deg; joints [-12.669, -27.452, 110.066, -16.731, -82.061, 51.349]
  MoveL 6086 to (509.44, 509.44, 13.1) mm, rotated rx 0 ry 90 rz 0 deg; joints [-12.677, -27.449, 110.048, -16.74, -82.047, 51.354]
  Set speed (120.0 mm/s)
  MoveL 6087 to (507.39, 502.51, 13.1) mm, rotated rx 0 ry 90 rz 0 deg; joints [-12.094, -27.521, 110.479, -16.138, -82.371, 51.181]
  Set speed (30.0 mm/s)
  Call Extruder(0.280)
  MoveL 6088 to (500.58, 509.32, 13.1) mm, rotated rx 0 ry 90 rz 0 deg; joints [-12.847, -27.623, 111.114, -16.878, -82.906, 51.114]
  Set speed (120.0 mm/s)
  MoveL 6089 to (499.42, 509.32, 13.1) mm, rotated rx 0 ry 90 rz 0 deg; joints [-12.872, -27.645, 111.252, -16.898, -83.018, 51.083]
  Set speed (30.0 mm/s)
  Call Extruder(0.360)
  MoveL 6090 to (490.68, 500.58, 13.1) mm, rotated rx 0 ry 90 rz 0 deg; joints [-12.247, -27.835, 112.519, -16.234, -84.033, 50.712]
  Set speed (120.0 mm/s)
  MoveL 6091 to (490.68, 499.42, 13.1) mm, rotated rx 0 ry 90 rz 0 deg; joints [-12.139, -27.839, 112.549, -16.125, -84.055, 50.696]
  Set speed (30.0 mm/s)
  Call Extruder(0.282)
  MoveL 6092 to (497.52, 492.58, 13.1) mm, rotated rx 0 ry 90 rz 0 deg; joints [-11.373, -27.745, 111.906, -15.371, -83.506, 50.773]
  MoveL 6093 to (497.64, 492.46, 13.1) mm, rotated rx 0 ry 90 rz 0 deg; joints [-11.359, -27.743, 111.895, -15.358, -83.496, 50.775]
  Set speed (120.0 mm/s)
  MoveL 6094 to (502.48, 492.58, 13.1) mm, rotated rx 0 ry 90 rz 0 deg; joints [-11.281, -27.655, 111.314, -15.295, -83.02, 50.898]
  Set speed (30.0 mm/s)
  Call Extruder(0.202)
  MoveL 6095 to (507.39, 497.49, 13.1) mm, rotated rx 0 ry 90 rz 0 deg; joints [-11.639, -27.541, 110.605, -15.675, -82.457, 51.098]
  MoveL 6096 to (507.51, 497.61, 13.1) mm, rotated rx 0 ry 90 rz 0 deg; joints [-11.647, -27.538, 110.587, -15.684, -82.443, 51.103]
  Set speed (120.0 mm/s)
  MoveL 6097 to (508.76, 498.86, 13.1) mm, rotated rx 0 ry 90 rz 0 deg; joints [-11.737, -27.509, 110.407, -15.78, -82.3, 51.155]
  Set speed (30.0 mm/s)
  Call Extruder(0.023)
  MoveL 6098 to (509.32, 499.42, 13.1) mm, rotated rx 0 ry 90 rz 0 deg; joints [-11.777, -27.495, 110.325, -15.823, -82.236, 51.179]
  Set speed (120.0 mm/s)
  MoveL 6099 to (507.64, 498.61, 13.1) mm, rotated rx 0 ry 90 rz 0 deg; joints [-11.735, -27.532, 110.547, -15.774, -82.413, 51.123]
  Set speed (1000.0 mm/s)
  MoveL 6100 to (507.64, 496.05, 13.1) mm, rotated rx 0 ry 90 rz 0 deg; joints [-11.503, -27.542, 110.61, -15.538, -82.457, 51.081]
  Set speed (1000.0 mm/s)
  MoveL 6101 to (509.32, 490.68, 13.1) mm, rotated rx 0 ry 90 rz 0 deg; joints [-10.985, -27.53, 110.537, -15.018, -82.381, 51.036]
  Set speed (30.0 mm/s)
  Call Extruder(0.767)
  MoveL 6102 to (490.68, 509.32, 13.1) mm, rotated rx 0 ry 90 rz 0 deg; joints [-13.056, -27.801, 112.288, -17.054, -83.865, 50.843]
  MoveL 6103 to (490.56, 509.44, 13.1) mm, rotated rx 0 ry 90 rz 0 deg; joints [-13.07, -27.803, 112.299, -17.067, -83.874, 50.841]
  Set speed (120.0 mm/s)
  MoveL 6104 to (502.71, 492.37, 13.1) mm, rotated rx 0 ry 90 rz 0 deg; joints [-11.258, -27.651, 111.291, -15.272, -83, 50.9]
  Set speed (1000.0 mm/s)
  MoveL 6105 to (502.64, 492.3, 13.1) mm, rotated rx 0 ry 90 rz 0 deg; joints [-11.253, -27.652, 111.301, -15.266, -83.008, 50.897]
  Set speed (15.0 mm/s)
  Call Extruder(0.010)
  MoveL 6106 to (502.64, 491.95, 13.1) mm, rotated rx 0 ry 90 rz 0 deg; joints [-11.221, -27.654, 111.309, -15.234, -83.014, 50.892]
  Call Extruder(0.035)
  MoveL 6107 to (502.64, 490.75, 13.1) mm, rotated rx 0 ry 90 rz 0 deg; joints [-11.111, -27.658, 111.338, -15.122, -83.034, 50.874]
  Call Extruder(0.010)
  MoveL 6108 to (502.64, 490.4, 13.1) mm, rotated rx 0 ry 90 rz 0 deg; joints [-11.079, -27.659, 111.346, -15.09, -83.04, 50.869]
  Call Extruder(0.007)
  MoveL 6109 to (502.99, 490.4, 13.1) mm, rotated rx 0 ry 90 rz 0 deg; joints [-11.072, -27.653, 111.304, -15.084, -83.006, 50.877]
  Call Extruder(0.192)
  MoveL 6110 to (509.6, 490.4, 13.1) mm, rotated rx 0 ry 90 rz 0 deg; joints [-10.955, -27.526, 110.509, -14.988, -82.358, 51.039]
  Call Extruder(0.165)
  MoveL 6111 to (509.6, 496.07, 13.1) mm, rotated rx 0 ry 90 rz 0 deg; joints [-11.469, -27.503, 110.374, -15.511, -82.265, 51.13]
  Call Extruder(0.056)
  MoveL 6112 to (507.67, 496.08, 13.1) mm, rotated rx 0 ry 90 rz 0 deg; joints [-11.505, -27.542, 110.606, -15.54, -82.453, 51.082]
  Call Extruder(0.063)
  MoveL 6113 to (507.67, 498.23, 13.1) mm, rotated rx 0 ry 90 rz 0 deg; joints [-11.7, -27.533, 110.553, -15.739, -82.417, 51.117]
  Call Extruder(0.010)
  MoveL 6114 to (507.67, 498.58, 13.1) mm, rotated rx 0 ry 90 rz 0 deg; joints [-11.732, -27.531, 110.544, -15.771, -82.411, 51.123]
  Call Extruder(0.007)
  MoveL 6115 to (508.02, 498.58, 13.1) mm, rotated rx 0 ry 90 rz 0 deg; joints [-11.725, -27.524, 110.502, -15.766, -82.377, 51.132]
  Call Extruder(0.046)
  MoveL 6116 to (509.6, 498.58, 13.1) mm, rotated rx 0 ry 90 rz 0 deg; joints [-11.696, -27.493, 110.312, -15.741, -82.223, 51.172]
  Call Extruder(0.057)
  MoveL 6117 to (509.6, 500.53, 13.1) mm, rotated rx 0 ry 90 rz 0 deg; joints [-11.872, -27.485, 110.263, -15.92, -82.19, 51.204]
  Call Extruder(0.046)
  MoveL 6118 to (508.02, 500.52, 13.1) mm, rotated rx 0 ry 90 rz 0 deg; joints [-11.902, -27.516, 110.453, -15.945, -82.344, 51.164]
  Call Extruder(0.010)
  MoveL 6119 to (507.67, 500.52, 13.1) mm, rotated rx 0 ry 90 rz 0 deg; joints [-11.908, -27.523, 110.496, -15.95, -82.378, 51.155]
  Call Extruder(0.007)
  MoveL 6120 to (507.67, 500.87, 13.1) mm, rotated rx 0 ry 90 rz 0 deg; joints [-11.94, -27.522, 110.487, -15.982, -82.372, 51.161]
  Call Extruder(0.062)
  MoveL 6121 to (507.67, 503.01, 13.1) mm, rotated rx 0 ry 90 rz 0 deg; joints [-12.133, -27.513, 110.432, -16.179, -82.334, 51.197]
  Call Extruder(0.056)
  MoveL 6122 to (509.6, 503.02, 13.1) mm, rotated rx 0 ry 90 rz 0 deg; joints [-12.096, -27.474, 110.199, -16.149, -82.147, 51.247]
  Call Extruder(0.192)
  MoveL 6123 to (509.6, 509.6, 13.1) mm, rotated rx 0 ry 90 rz 0 deg; joints [-12.688, -27.445, 110.025, -16.752, -82.029, 51.361]
  Call Extruder(0.559)
  MoveL 6124 to (490.4, 509.6, 13.1) mm, rotated rx 0 ry 90 rz 0 deg; joints [-13.088, -27.805, 112.313, -17.085, -83.886, 50.839]
  MoveL 6125 to (490.4, 490.4, 13.1) mm, rotated rx 0 ry 90 rz 0 deg; joints [-11.303, -27.875, 112.803, -15.279, -84.244, 50.563]
  Call Extruder(0.168)
  MoveL 6126 to (496.16, 490.4, 13.1) mm, rotated rx 0 ry 90 rz 0 deg; joints [-11.196, -27.777, 112.12, -15.188, -83.677, 50.708]
  Call Extruder(0.010)
  MoveL 6127 to (496.51, 490.4, 13.1) mm, rotated rx 0 ry 90 rz 0 deg; joints [-11.19, -27.771, 112.078, -15.183, -83.643, 50.717]
  Call Extruder(0.007)
  MoveL 6128 to (496.51, 490.75, 13.1) mm, rotated rx 0 ry 90 rz 0 deg; joints [-11.222, -27.769, 112.07, -15.216, -83.637, 50.722]
  Call Extruder(0.035)
  MoveL 6129 to (496.51, 491.95, 13.1) mm, rotated rx 0 ry 90 rz 0 deg; joints [-11.334, -27.765, 112.042, -15.328, -83.617, 50.739]
  Call Extruder(0.010)
  MoveL 6130 to (496.51, 492.3, 13.1) mm, rotated rx 0 ry 90 rz 0 deg; joints [-11.366, -27.764, 112.033, -15.361, -83.611, 50.744]
  Call Extruder(0.007)
  MoveL 6131 to (496.86, 492.3, 13.1) mm, rotated rx 0 ry 90 rz 0 deg; joints [-11.36, -27.758, 111.992, -15.356, -83.576, 50.753]
  Call Extruder(0.061)
  MoveL 6132 to (498.97, 492.3, 13.1) mm, rotated rx 0 ry 90 rz 0 deg; joints [-11.32, -27.72, 111.741, -15.323, -83.369, 50.806]
  Call Extruder(0.055)
  MoveL 6133 to (498.97, 490.4, 13.1) mm, rotated rx 0 ry 90 rz 0 deg; joints [-11.145, -27.727, 111.785, -15.145, -83.401, 50.778]
  Call Extruder(0.036)
  MoveL 6134 to (500.22, 490.4, 13.1) mm, rotated rx 0 ry 90 rz 0 deg; joints [-11.122, -27.704, 111.636, -15.126, -83.278, 50.809]
  Call Extruder(0.055)
  MoveL 6135 to (500.22, 492.3, 13.1) mm, rotated rx 0 ry 90 rz 0 deg; joints [-11.297, -27.697, 111.591, -15.303, -83.246, 50.837]
  Call Extruder(0.060)
  MoveL 6136 to (502.29, 492.3, 13.1) mm, rotated rx 0 ry 90 rz 0 deg; joints [-11.259, -27.659, 111.343, -15.272, -83.043, 50.889]
  Call Extruder(0.007)
  MoveL 6137 to (502.64, 492.3, 13.1) mm, rotated rx 0 ry 90 rz 0 deg; joints [-11.253, -27.652, 111.301, -15.266, -83.008, 50.897]
  Set speed (120.0 mm/s)
  MoveL 6138 to (502.64, 491.95, 13.1) mm, rotated rx 0 ry 90 rz 0 deg; joints [-11.221, -27.654, 111.309, -15.234, -83.014, 50.892]
  Set speed (1000.0 mm/s)
  MoveL 6139 to (502.64, 491.9, 13.1) mm, rotated rx 0 ry 90 rz 0 deg; joints [-11.216, -27.654, 111.31, -15.229, -83.015, 50.891]
  Set speed (1000.0 mm/s)
  MoveL 6140 to (502.74, 491.9, 13.1) mm, rotated rx 0 ry 90 rz 0 deg; joints [-11.214, -27.652, 111.298, -15.228, -83.005, 50.894]
  Set speed (1000.0 mm/s)
  MoveL 6141 to (500.19, 492.33, 13.1) mm, rotated rx 0 ry 90 rz 0 deg; joints [-11.3, -27.698, 111.594, -15.306, -83.249, 50.837]
  Set speed (1000.0 mm/s)
  MoveL 6142 to (499.59, 491.67, 13.1) mm, rotated rx 0 ry 90 rz 0 deg; joints [-11.251, -27.711, 111.681, -15.254, -83.318, 50.812]
  Set speed (15.0 mm/s)
  Call Extruder(0.008)
  MoveL 6143 to (499.59, 492.17, 13.1) mm, rotated rx 0 ry 90 rz 0 deg; joints [-11.297, -27.709, 111.669, -15.3, -83.31, 50.819]
  Call Extruder(0.006)
  MoveL 6144 to (499.45, 492.52, 13.1) mm, rotated rx 0 ry 90 rz 0 deg; joints [-11.332, -27.71, 111.677, -15.336, -83.318, 50.821]
  Call Extruder(0.029)
  MoveL 6145 to (499.76, 490.85, 13.1) mm, rotated rx 0 ry 90 rz 0 deg; joints [-11.172, -27.711, 111.68, -15.175, -83.315, 50.804]
  Set speed (120.0 mm/s)
  MoveL 6146 to (499.67, 490.98, 13.1) mm, rotated rx 0 ry 90 rz 0 deg; joints [-11.185, -27.712, 111.688, -15.188, -83.323, 50.804]
  Set speed (1000.0 mm/s)
  MoveL 6147 to (498.99, 492.33, 13.1) mm, rotated rx 0 ry 90 rz 0 deg; joints [-11.322, -27.719, 111.737, -15.325, -83.366, 50.807]
  Set speed (1000.0 mm/s)
  MoveL 6148 to (496.48, 492.33, 13.1) mm, rotated rx 0 ry 90 rz 0 deg; joints [-11.369, -27.764, 112.036, -15.364, -83.613, 50.744]
  Set speed (1000.0 mm/s)
  MoveL 6149 to (490.68, 490.68, 13.1) mm, rotated rx 0 ry 90 rz 0 deg; joints [-11.324, -27.869, 112.763, -15.301, -84.212, 50.574]
  Set speed (1000.0 mm/s)
  MoveL 6150 to (490.68, 490.68, 13.2) mm, rotated rx 0 ry 90 rz 0 deg; joints [-11.324, -27.88, 112.768, -15.301, -84.207, 50.575]
  Set speed (30.0 mm/s)
  Call Extruder(0.767)
  MoveL 6151 to (509.32, 509.32, 13.2) mm, rotated rx 0 ry 90 rz 0 deg; joints [-12.669, -27.462, 110.071, -16.731, -82.056, 51.35]
  MoveL 6152 to (509.44, 509.44, 13.2) mm, rotated rx 0 ry 90 rz 0 deg; joints [-12.677, -27.459, 110.053, -16.74, -82.042, 51.356]
  Set speed (120.0 mm/s)
  MoveL 6153 to (507.39, 502.51, 13.2) mm, rotated rx 0 ry 90 rz 0 deg; joints [-12.094, -27.531, 110.484, -16.138, -82.365, 51.182]
  Set speed (30.0 mm/s)
  Call Extruder(0.280)
  MoveL 6154 to (500.58, 509.32, 13.2) mm, rotated rx 0 ry 90 rz 0 deg; joints [-12.847, -27.634, 111.119, -16.878, -82.901, 51.116]
  Set speed (120.0 mm/s)
  MoveL 6155 to (499.42, 509.32, 13.2) mm, rotated rx 0 ry 90 rz 0 deg; joints [-12.872, -27.655, 111.257, -16.898, -83.013, 51.084]
  Set speed (30.0 mm/s)
  Call Extruder(0.360)
  MoveL 6156 to (490.68, 500.58, 13.2) mm, rotated rx 0 ry 90 rz 0 deg; joints [-12.247, -27.845, 112.524, -16.234, -84.028, 50.714]
  Set speed (120.0 mm/s)
  MoveL 6157 to (490.68, 499.42, 13.2) mm, rotated rx 0 ry 90 rz 0 deg; joints [-12.139, -27.85, 112.554, -16.125, -84.049, 50.697]
  Set speed (30.0 mm/s)
  Call Extruder(0.281)
  MoveL 6158 to (497.52, 492.58, 13.2) mm, rotated rx 0 ry 90 rz 0 deg; joints [-11.373, -27.756, 111.911, -15.372, -83.501, 50.775]
  MoveL 6159 to (497.64, 492.46, 13.2) mm, rotated rx 0 ry 90 rz 0 deg; joints [-11.36, -27.754, 111.9, -15.358, -83.491, 50.776]
  Set speed (120.0 mm/s)
  MoveL 6160 to (502.48, 492.58, 13.2) mm, rotated rx 0 ry 90 rz 0 deg; joints [-11.282, -27.665, 111.319, -15.295, -83.015, 50.899]
  Set speed (30.0 mm/s)
  Call Extruder(0.202)
  MoveL 6161 to (507.39, 497.49, 13.2) mm, rotated rx 0 ry 90 rz 0 deg; joints [-11.639, -27.552, 110.61, -15.675, -82.452, 51.099]
  MoveL 6162 to (507.51, 497.61, 13.2) mm, rotated rx 0 ry 90 rz 0 deg; joints [-11.647, -27.549, 110.593, -15.685, -82.438, 51.105]
  Set speed (120.0 mm/s)
  MoveL 6163 to (508.7, 498.8, 13.2) mm, rotated rx 0 ry 90 rz 0 deg; joints [-11.733, -27.521, 110.42, -15.776, -82.302, 51.154]
  Set speed (30.0 mm/s)
  Call Extruder(0.026)
  MoveL 6164 to (509.32, 499.42, 13.2) mm, rotated rx 0 ry 90 rz 0 deg; joints [-11.777, -27.506, 110.33, -15.823, -82.231, 51.18]
  Set speed (120.0 mm/s)
  MoveL 6165 to (507.64, 498.55, 13.2) mm, rotated rx 0 ry 90 rz 0 deg; joints [-11.73, -27.543, 110.554, -15.769, -82.409, 51.123]
  Set speed (1000.0 mm/s)
  MoveL 6166 to (507.64, 495.99, 13.2) mm, rotated rx 0 ry 90 rz 0 deg; joints [-11.498, -27.553, 110.617, -15.533, -82.453, 51.081]
  Set speed (1000.0 mm/s)
  MoveL 6167 to (509.32, 490.68, 13.2) mm, rotated rx 0 ry 90 rz 0 deg; joints [-10.985, -27.541, 110.542, -15.018, -82.376, 51.038]
  Set speed (30.0 mm/s)
  Call Extruder(0.767)
  MoveL 6168 to (490.68, 509.32, 13.2) mm, rotated rx 0 ry 90 rz 0 deg; joints [-13.056, -27.812, 112.293, -17.054, -83.86, 50.845]
  MoveL 6169 to (490.56, 509.44, 13.2) mm, rotated rx 0 ry 90 rz 0 deg; joints [-13.07, -27.814, 112.304, -17.068, -83.869, 50.843]
  Set speed (120.0 mm/s)
  MoveL 6170 to (502.78, 492.37, 13.2) mm, rotated rx 0 ry 90 rz 0 deg; joints [-11.257, -27.66, 111.288, -15.271, -82.989, 50.903]
  Set speed (1000.0 mm/s)
  MoveL 6171 to (502.71, 492.3, 13.2) mm, rotated rx 0 ry 90 rz 0 deg; joints [-11.252, -27.662, 111.298, -15.266, -82.997, 50.9]
  Set speed (15.0 mm/s)
  Call Extruder(0.010)
  MoveL 6172 to (502.71, 491.95, 13.2) mm, rotated rx 0 ry 90 rz 0 deg; joints [-11.22, -27.663, 111.307, -15.233, -83.003, 50.895]
  Call Extruder(0.035)
  MoveL 6173 to (502.71, 490.75, 13.2) mm, rotated rx 0 ry 90 rz 0 deg; joints [-11.11, -27.668, 111.335, -15.121, -83.023, 50.877]
  Call Extruder(0.010)
  MoveL 6174 to (502.71, 490.4, 13.2) mm, rotated rx 0 ry 90 rz 0 deg; joints [-11.077, -27.669, 111.343, -15.089, -83.029, 50.872]
  Call Extruder(0.007)
  MoveL 6175 to (503.06, 490.4, 13.2) mm, rotated rx 0 ry 90 rz 0 deg; joints [-11.071, -27.662, 111.301, -15.084, -82.994, 50.88]
  Call Extruder(0.190)
  MoveL 6176 to (509.6, 490.4, 13.2) mm, rotated rx 0 ry 90 rz 0 deg; joints [-10.955, -27.536, 110.515, -14.989, -82.353, 51.04]
  Call Extruder(0.163)
  MoveL 6177 to (509.6, 496.01, 13.2) mm, rotated rx 0 ry 90 rz 0 deg; joints [-11.464, -27.514, 110.38, -15.506, -82.261, 51.131]
  Call Extruder(0.056)
  MoveL 6178 to (507.67, 496.02, 13.2) mm, rotated rx 0 ry 90 rz 0 deg; joints [-11.5, -27.552, 110.613, -15.535, -82.449, 51.083]
  Call Extruder(0.063)
  MoveL 6179 to (507.67, 498.17, 13.2) mm, rotated rx 0 ry 90 rz 0 deg; joints [-11.695, -27.544, 110.56, -15.734, -82.413, 51.118]
  Call Extruder(0.010)
  MoveL 6180 to (507.67, 498.52, 13.2) mm, rotated rx 0 ry 90 rz 0 deg; joints [-11.727, -27.542, 110.551, -15.766, -82.407, 51.123]
  Call Extruder(0.007)
  MoveL 6181 to (508.02, 498.52, 13.2) mm, rotated rx 0 ry 90 rz 0 deg; joints [-11.72, -27.535, 110.509, -15.76, -82.373, 51.132]
  Call Extruder(0.036)
  MoveL 6182 to (509.25, 498.52, 13.2) mm, rotated rx 0 ry 90 rz 0 deg; joints [-11.697, -27.511, 110.361, -15.742, -82.253, 51.163]
  Call Extruder(0.010)
  MoveL 6183 to (509.6, 498.52, 13.2) mm, rotated rx 0 ry 90 rz 0 deg; joints [-11.691, -27.504, 110.318, -15.736, -82.219, 51.172]
  Call Extruder(0.007)
  MoveL 6184 to (509.6, 498.87, 13.2) mm, rotated rx 0 ry 90 rz 0 deg; joints [-11.722, -27.502, 110.31, -15.768, -82.213, 51.178]
  Call Extruder(0.040)
  MoveL 6185 to (509.6, 500.23, 13.2) mm, rotated rx 0 ry 90 rz 0 deg; joints [-11.845, -27.497, 110.275, -15.894, -82.19, 51.201]
  Call Extruder(0.010)
  MoveL 6186 to (509.6, 500.58, 13.2) mm, rotated rx 0 ry 90 rz 0 deg; joints [-11.877, -27.495, 110.267, -15.926, -82.184, 51.207]
  Call Extruder(0.007)
  MoveL 6187 to (509.25, 500.58, 13.2) mm, rotated rx 0 ry 90 rz 0 deg; joints [-11.883, -27.502, 110.309, -15.931, -82.218, 51.198]
  Call Extruder(0.036)
  MoveL 6188 to (508.02, 500.58, 13.2) mm, rotated rx 0 ry 90 rz 0 deg; joints [-11.907, -27.527, 110.457, -15.95, -82.338, 51.166]
  Call Extruder(0.010)
  MoveL 6189 to (507.67, 500.58, 13.2) mm, rotated rx 0 ry 90 rz 0 deg; joints [-11.913, -27.534, 110.499, -15.956, -82.372, 51.157]
  Call Extruder(0.007)
  MoveL 6190 to (507.67, 500.93, 13.2) mm, rotated rx 0 ry 90 rz 0 deg; joints [-11.945, -27.532, 110.49, -15.988, -82.366, 51.163]
  Call Extruder(0.062)
  MoveL 6191 to (507.67, 503.07, 13.2) mm, rotated rx 0 ry 90 rz 0 deg; joints [-12.138, -27.523, 110.436, -16.184, -82.328, 51.199]
  Call Extruder(0.056)
  MoveL 6192 to (509.6, 503.07, 13.2) mm, rotated rx 0 ry 90 rz 0 deg; joints [-12.101, -27.484, 110.203, -16.154, -82.141, 51.249]
  Call Extruder(0.190)
  MoveL 6193 to (509.6, 509.6, 13.2) mm, rotated rx 0 ry 90 rz 0 deg; joints [-12.688, -27.455, 110.03, -16.752, -82.024, 51.363]
  Call Extruder(0.559)
  MoveL 6194 to (490.4, 509.6, 13.2) mm, rotated rx 0 ry 90 rz 0 deg; joints [-13.088, -27.816, 112.318, -17.085, -83.881, 50.841]
  MoveL 6195 to (490.4, 490.4, 13.2) mm, rotated rx 0 ry 90 rz 0 deg; joints [-11.303, -27.885, 112.808, -15.279, -84.239, 50.565]
  Call Extruder(0.166)
  MoveL 6196 to (496.1, 490.4, 13.2) mm, rotated rx 0 ry 90 rz 0 deg; joints [-11.197, -27.788, 112.132, -15.189, -83.678, 50.708]
  Call Extruder(0.010)
  MoveL 6197 to (496.45, 490.4, 13.2) mm, rotated rx 0 ry 90 rz 0 deg; joints [-11.191, -27.782, 112.09, -15.184, -83.643, 50.717]
  Call Extruder(0.007)
  MoveL 6198 to (496.45, 490.75, 13.2) mm, rotated rx 0 ry 90 rz 0 deg; joints [-11.223, -27.781, 112.082, -15.217, -83.637, 50.722]
  Call Extruder(0.035)
  MoveL 6199 to (496.45, 491.95, 13.2) mm, rotated rx 0 ry 90 rz 0 deg; joints [-11.335, -27.777, 112.054, -15.329, -83.617, 50.739]
  Call Extruder(0.010)
  MoveL 6200 to (496.45, 492.3, 13.2) mm, rotated rx 0 ry 90 rz 0 deg; joints [-11.367, -27.776, 112.045, -15.362, -83.611, 50.744]
  Call Extruder(0.007)
  MoveL 6201 to (496.8, 492.3, 13.2) mm, rotated rx 0 ry 90 rz 0 deg; joints [-11.361, -27.769, 112.004, -15.357, -83.576, 50.753]
  Call Extruder(0.061)
  MoveL 6202 to (498.91, 492.3, 13.2) mm, rotated rx 0 ry 90 rz 0 deg; joints [-11.322, -27.732, 111.752, -15.324, -83.37, 50.806]
  Call Extruder(0.055)
  MoveL 6203 to (498.91, 490.4, 13.2) mm, rotated rx 0 ry 90 rz 0 deg; joints [-11.146, -27.738, 111.797, -15.146, -83.402, 50.778]
  Call Extruder(0.040)
  MoveL 6204 to (500.28, 490.4, 13.2) mm, rotated rx 0 ry 90 rz 0 deg; joints [-11.121, -27.714, 111.634, -15.125, -83.267, 50.812]
  Call Extruder(0.055)
  MoveL 6205 to (500.28, 492.3, 13.2) mm, rotated rx 0 ry 90 rz 0 deg; joints [-11.296, -27.707, 111.588, -15.303, -83.235, 50.84]
  Call Extruder(0.060)
  MoveL 6206 to (502.36, 492.3, 13.2) mm, rotated rx 0 ry 90 rz 0 deg; joints [-11.258, -27.668, 111.34, -15.271, -83.031, 50.892]
  Call Extruder(0.007)
  MoveL 6207 to (502.71, 492.3, 13.2) mm, rotated rx 0 ry 90 rz 0 deg; joints [-11.252, -27.662, 111.298, -15.266, -82.997, 50.9]
  Set speed (120.0 mm/s)
  MoveL 6208 to (502.71, 491.95, 13.2) mm, rotated rx 0 ry 90 rz 0 deg; joints [-11.22, -27.663, 111.307, -15.233, -83.003, 50.895]
  Set speed (1000.0 mm/s)
  MoveL 6209 to (502.71, 491.9, 13.2) mm, rotated rx 0 ry 90 rz 0 deg; joints [-11.215, -27.663, 111.308, -15.228, -83.004, 50.894]
  Set speed (1000.0 mm/s)
  MoveL 6210 to (502.81, 491.9, 13.2) mm, rotated rx 0 ry 90 rz 0 deg; joints [-11.213, -27.661, 111.296, -15.227, -82.994, 50.897]
  Set speed (1000.0 mm/s)
  MoveL 6211 to (500.25, 492.33, 13.2) mm, rotated rx 0 ry 90 rz 0 deg; joints [-11.299, -27.707, 111.591, -15.306, -83.237, 50.84]
  Set speed (1000.0 mm/s)
  MoveL 6212 to (499.95, 491.98, 13.2) mm, rotated rx 0 ry 90 rz 0 deg; joints [-11.273, -27.714, 111.636, -15.278, -83.273, 50.827]
  Set speed (15.0 mm/s)
  Call Extruder(0.015)
  MoveL 6213 to (499.24, 492.69, 13.2) mm, rotated rx 0 ry 90 rz 0 deg; joints [-11.351, -27.724, 111.703, -15.355, -83.33, 50.82]
  Set speed (120.0 mm/s)
  MoveL 6214 to (499.24, 492.19, 13.2) mm, rotated rx 0 ry 90 rz 0 deg; joints [-11.306, -27.726, 111.716, -15.309, -83.339, 50.812]
  Set speed (15.0 mm/s)
  Call Extruder(0.015)
  MoveL 6215 to (499.95, 491.48, 13.2) mm, rotated rx 0 ry 90 rz 0 deg; joints [-11.227, -27.716, 111.648, -15.231, -83.281, 50.82]
  Set speed (120.0 mm/s)
  MoveL 6216 to (499.95, 490.99, 13.2) mm, rotated rx 0 ry 90 rz 0 deg; joints [-11.182, -27.718, 111.659, -15.185, -83.29, 50.812]
  Set speed (15.0 mm/s)
  Call Extruder(0.015)
  MoveL 6217 to (499.24, 491.7, 13.2) mm, rotated rx 0 ry 90 rz 0 deg; joints [-11.26, -27.728, 111.727, -15.263, -83.347, 50.805]
  Set speed (120.0 mm/s)
  MoveL 6218 to (499.48, 490.97, 13.2) mm, rotated rx 0 ry 90 rz 0 deg; joints [-11.188, -27.726, 111.716, -15.19, -83.336, 50.8]
  Set speed (15.0 mm/s)
  Call Extruder(0.014)
  MoveL 6219 to (499.84, 492.58, 13.2) mm, rotated rx 0 ry 90 rz 0 deg; joints [-11.33, -27.714, 111.634, -15.335, -83.273, 50.833]
  Set speed (120.0 mm/s)
  MoveL 6220 to (499.79, 492.8, 13.2) mm, rotated rx 0 ry 90 rz 0 deg; joints [-11.351, -27.714, 111.636, -15.356, -83.275, 50.835]
  Set speed (1000.0 mm/s)
  MoveL 6221 to (496.42, 492.33, 13.2) mm, rotated rx 0 ry 90 rz 0 deg; joints [-11.37, -27.776, 112.048, -15.365, -83.613, 50.744]
  Set speed (1000.0 mm/s)
  MoveL 6222 to (490.68, 490.68, 13.2) mm, rotated rx 0 ry 90 rz 0 deg; joints [-11.324, -27.88, 112.768, -15.301, -84.207, 50.575]
  Set speed (1000.0 mm/s)
  MoveL 6223 to (490.68, 490.68, 13.3) mm, rotated rx 0 ry 90 rz 0 deg; joints [-11.324, -27.891, 112.774, -15.301, -84.201, 50.577]
  Set speed (30.0 mm/s)
  Call Extruder(0.767)
  MoveL 6224 to (509.32, 509.32, 13.3) mm, rotated rx 0 ry 90 rz 0 deg; joints [-12.669, -27.473, 110.077, -16.731, -82.051, 51.352]
  MoveL 6225 to (509.44, 509.44, 13.3) mm, rotated rx 0 ry 90 rz 0 deg; joints [-12.677, -27.47, 110.058, -16.74, -82.037, 51.357]
  Set speed (120.0 mm/s)
  MoveL 6226 to (507.39, 502.51, 13.3) mm, rotated rx 0 ry 90 rz 0 deg; joints [-12.094, -27.542, 110.489, -16.138, -82.36, 51.184]
  Set speed (30.0 mm/s)
  Call Extruder(0.280)
  MoveL 6227 to (500.58, 509.32, 13.3) mm, rotated rx 0 ry 90 rz 0 deg; joints [-12.847, -27.644, 111.124, -16.878, -82.896, 51.118]
  Set speed (120.0 mm/s)
  MoveL 6228 to (499.42, 509.32, 13.3) mm, rotated rx 0 ry 90 rz 0 deg; joints [-12.872, -27.666, 111.262, -16.898, -83.008, 51.086]
  Set speed (30.0 mm/s)
  Call Extruder(0.360)
  MoveL 6229 to (490.68, 500.58, 13.3) mm, rotated rx 0 ry 90 rz 0 deg; joints [-12.247, -27.856, 112.529, -16.235, -84.022, 50.715]
  Set speed (120.0 mm/s)
  MoveL 6230 to (490.68, 499.42, 13.3) mm, rotated rx 0 ry 90 rz 0 deg; joints [-12.139, -27.86, 112.559, -16.125, -84.044, 50.699]
  Set speed (30.0 mm/s)
  Call Extruder(0.281)
  MoveL 6231 to (497.52, 492.58, 13.3) mm, rotated rx 0 ry 90 rz 0 deg; joints [-11.373, -27.766, 111.917, -15.372, -83.496, 50.776]
  MoveL 6232 to (497.64, 492.46, 13.3) mm, rotated rx 0 ry 90 rz 0 deg; joints [-11.359, -27.764, 111.905, -15.358, -83.486, 50.778]
  Set speed (120.0 mm/s)
  MoveL 6233 to (499.13, 490.97, 13.3) mm, rotated rx 0 ry 90 rz 0 deg; joints [-11.194, -27.743, 111.763, -15.196, -83.365, 50.793]
  Set speed (30.0 mm/s)
  Call Extruder(0.012)
  MoveL 6234 to (499.42, 490.68, 13.3) mm, rotated rx 0 ry 90 rz 0 deg; joints [-11.163, -27.739, 111.735, -15.165, -83.342, 50.796]
  Set speed (120.0 mm/s)
  MoveL 6235 to (500.32, 492.33, 13.3) mm, rotated rx 0 ry 90 rz 0 deg; joints [-11.298, -27.717, 111.589, -15.305, -83.226, 50.843]
  Set speed (1000.0 mm/s)
  MoveL 6236 to (502.48, 492.58, 13.3) mm, rotated rx 0 ry 90 rz 0 deg; joints [-11.282, -27.676, 111.324, -15.295, -83.009, 50.9]
  Set speed (30.0 mm/s)
  Call Extruder(0.202)
  MoveL 6237 to (507.39, 497.49, 13.3) mm, rotated rx 0 ry 90 rz 0 deg; joints [-11.639, -27.562, 110.615, -15.675, -82.447, 51.101]
  MoveL 6238 to (507.51, 497.61, 13.3) mm, rotated rx 0 ry 90 rz 0 deg; joints [-11.647, -27.559, 110.598, -15.685, -82.433, 51.106]
  Set speed (120.0 mm/s)
  MoveL 6239 to (508.64, 498.74, 13.3) mm, rotated rx 0 ry 90 rz 0 deg; joints [-11.728, -27.532, 110.434, -15.771, -82.303, 51.153]
  Set speed (30.0 mm/s)
  Call Extruder(0.028)
  MoveL 6240 to (509.32, 499.42, 13.3) mm, rotated rx 0 ry 90 rz 0 deg; joints [-11.777, -27.516, 110.335, -15.824, -82.226, 51.182]
  Set speed (120.0 mm/s)
  MoveL 6241 to (507.64, 498.49, 13.3) mm, rotated rx 0 ry 90 rz 0 deg; joints [-11.725, -27.553, 110.56, -15.764, -82.405, 51.124]
  Set speed (1000.0 mm/s)
  MoveL 6242 to (507.64, 495.93, 13.3) mm, rotated rx 0 ry 90 rz 0 deg; joints [-11.492, -27.564, 110.623, -15.527, -82.448, 51.082]
  Set speed (1000.0 mm/s)
  MoveL 6243 to (509.32, 490.68, 13.3) mm, rotated rx 0 ry 90 rz 0 deg; joints [-10.985, -27.551, 110.547, -15.018, -82.371, 51.039]
  Set speed (30.0 mm/s)
  Call Extruder(0.767)
  MoveL 6244 to (490.68, 509.32, 13.3) mm, rotated rx 0 ry 90 rz 0 deg; joints [-13.056, -27.823, 112.298, -17.054, -83.855, 50.846]
  MoveL 6245 to (490.56, 509.44, 13.3) mm, rotated rx 0 ry 90 rz 0 deg; joints [-13.07, -27.824, 112.309, -17.068, -83.864, 50.845]
  Set speed (120.0 mm/s)
  MoveL 6246 to (502.84, 492.37, 13.3) mm, rotated rx 0 ry 90 rz 0 deg; joints [-11.256, -27.67, 111.286, -15.27, -82.977, 50.906]
  Set speed (1000.0 mm/s)
  MoveL 6247 to (502.77, 492.3, 13.3) mm, rotated rx 0 ry 90 rz 0 deg; joints [-11.251, -27.671, 111.296, -15.265, -82.985, 50.903]
  Set speed (15.0 mm/s)
  Call Extruder(0.010)
  MoveL 6248 to (502.77, 491.95, 13.3) mm, rotated rx 0 ry 90 rz 0 deg; joints [-11.218, -27.672, 111.304, -15.232, -82.991, 50.898]
  Call Extruder(0.035)
  MoveL 6249 to (502.77, 490.75, 13.3) mm, rotated rx 0 ry 90 rz 0 deg; joints [-11.108, -27.677, 111.333, -15.121, -83.011, 50.88]
  Call Extruder(0.010)
  MoveL 6250 to (502.77, 490.4, 13.3) mm, rotated rx 0 ry 90 rz 0 deg; joints [-11.076, -27.678, 111.341, -15.088, -83.017, 50.875]
  Call Extruder(0.007)
  MoveL 6251 to (503.12, 490.4, 13.3) mm, rotated rx 0 ry 90 rz 0 deg; joints [-11.07, -27.672, 111.299, -15.083, -82.983, 50.883]
  Call Extruder(0.189)
  MoveL 6252 to (509.6, 490.4, 13.3) mm, rotated rx 0 ry 90 rz 0 deg; joints [-10.955, -27.547, 110.52, -14.989, -82.347, 51.041]
  Call Extruder(0.162)
  MoveL 6253 to (509.6, 495.95, 13.3) mm, rotated rx 0 ry 90 rz 0 deg; joints [-11.459, -27.525, 110.387, -15.501, -82.257, 51.131]
  Call Extruder(0.056)
  MoveL 6254 to (507.67, 495.96, 13.3) mm, rotated rx 0 ry 90 rz 0 deg; joints [-11.494, -27.563, 110.619, -15.53, -82.445, 51.083]
  Call Extruder(0.063)
  MoveL 6255 to (507.67, 498.11, 13.3) mm, rotated rx 0 ry 90 rz 0 deg; joints [-11.69, -27.554, 110.566, -15.728, -82.409, 51.118]
  Call Extruder(0.010)
  MoveL 6256 to (507.67, 498.46, 13.3) mm, rotated rx 0 ry 90 rz 0 deg; joints [-11.721, -27.553, 110.558, -15.761, -82.403, 51.124]
  Call Extruder(0.007)
  MoveL 6257 to (508.02, 498.46, 13.3) mm, rotated rx 0 ry 90 rz 0 deg; joints [-11.715, -27.546, 110.515, -15.755, -82.369, 51.133]
  Call Extruder(0.036)
  MoveL 6258 to (509.25, 498.46, 13.3) mm, rotated rx 0 ry 90 rz 0 deg; joints [-11.692, -27.521, 110.367, -15.736, -82.249, 51.164]
  Call Extruder(0.010)
  MoveL 6259 to (509.6, 498.46, 13.3) mm, rotated rx 0 ry 90 rz 0 deg; joints [-11.685, -27.514, 110.325, -15.731, -82.215, 51.173]
  Call Extruder(0.007)
  MoveL 6260 to (509.6, 498.81, 13.3) mm, rotated rx 0 ry 90 rz 0 deg; joints [-11.717, -27.513, 110.316, -15.763, -82.209, 51.179]
  Call Extruder(0.043)
  MoveL 6261 to (509.6, 500.29, 13.3) mm, rotated rx 0 ry 90 rz 0 deg; joints [-11.85, -27.507, 110.279, -15.899, -82.184, 51.203]
  Call Extruder(0.010)
  MoveL 6262 to (509.6, 500.64, 13.3) mm, rotated rx 0 ry 90 rz 0 deg; joints [-11.882, -27.505, 110.27, -15.931, -82.178, 51.209]
  Call Extruder(0.007)
  MoveL 6263 to (509.25, 500.64, 13.3) mm, rotated rx 0 ry 90 rz 0 deg; joints [-11.888, -27.512, 110.312, -15.936, -82.212, 51.2]
  Call Extruder(0.036)
  MoveL 6264 to (508.02, 500.63, 13.3) mm, rotated rx 0 ry 90 rz 0 deg; joints [-11.912, -27.537, 110.461, -15.955, -82.331, 51.169]
  Call Extruder(0.010)
  MoveL 6265 to (507.67, 500.63, 13.3) mm, rotated rx 0 ry 90 rz 0 deg; joints [-11.918, -27.544, 110.503, -15.961, -82.366, 51.16]
  Call Extruder(0.007)
  MoveL 6266 to (507.67, 500.98, 13.3) mm, rotated rx 0 ry 90 rz 0 deg; joints [-11.95, -27.542, 110.494, -15.993, -82.359, 51.166]
  Call Extruder(0.062)
  MoveL 6267 to (507.67, 503.12, 13.3) mm, rotated rx 0 ry 90 rz 0 deg; joints [-12.144, -27.533, 110.439, -16.19, -82.322, 51.202]
  Call Extruder(0.056)
  MoveL 6268 to (509.6, 503.13, 13.3) mm, rotated rx 0 ry 90 rz 0 deg; joints [-12.106, -27.495, 110.206, -16.16, -82.134, 51.252]
  Call Extruder(0.188)
  MoveL 6269 to (509.6, 509.6, 13.3) mm, rotated rx 0 ry 90 rz 0 deg; joints [-12.688, -27.466, 110.035, -16.752, -82.019, 51.364]
  Call Extruder(0.559)
  MoveL 6270 to (490.4, 509.6, 13.3) mm, rotated rx 0 ry 90 rz 0 deg; joints [-13.088, -27.826, 112.323, -17.085, -83.876, 50.843]
  MoveL 6271 to (490.4, 490.4, 13.3) mm, rotated rx 0 ry 90 rz 0 deg; joints [-11.303, -27.896, 112.813, -15.279, -84.234, 50.566]
  Call Extruder(0.164)
  MoveL 6272 to (496.04, 490.4, 13.3) mm, rotated rx 0 ry 90 rz 0 deg; joints [-11.198, -27.8, 112.144, -15.19, -83.678, 50.708]
  Call Extruder(0.010)
  MoveL 6273 to (496.39, 490.4, 13.3) mm, rotated rx 0 ry 90 rz 0 deg; joints [-11.192, -27.794, 112.102, -15.185, -83.644, 50.717]
  Call Extruder(0.007)
  MoveL 6274 to (496.39, 490.75, 13.3) mm, rotated rx 0 ry 90 rz 0 deg; joints [-11.224, -27.793, 112.094, -15.218, -83.638, 50.722]
  Call Extruder(0.035)
  MoveL 6275 to (496.39, 491.95, 13.3) mm, rotated rx 0 ry 90 rz 0 deg; joints [-11.336, -27.788, 112.066, -15.33, -83.617, 50.739]
  Call Extruder(0.010)
  MoveL 6276 to (496.39, 492.3, 13.3) mm, rotated rx 0 ry 90 rz 0 deg; joints [-11.368, -27.787, 112.057, -15.363, -83.611, 50.744]
  Call Extruder(0.007)
  MoveL 6277 to (496.74, 492.3, 13.3) mm, rotated rx 0 ry 90 rz 0 deg; joints [-11.362, -27.781, 112.015, -15.358, -83.577, 50.753]
  Call Extruder(0.061)
  MoveL 6278 to (498.85, 492.3, 13.3) mm, rotated rx 0 ry 90 rz 0 deg; joints [-11.323, -27.743, 111.764, -15.325, -83.37, 50.806]
  Call Extruder(0.055)
  MoveL 6279 to (498.85, 490.4, 13.3) mm, rotated rx 0 ry 90 rz 0 deg; joints [-11.147, -27.75, 111.809, -15.147, -83.402, 50.778]
  Call Extruder(0.043)
  MoveL 6280 to (500.34, 490.4, 13.3) mm, rotated rx 0 ry 90 rz 0 deg; joints [-11.12, -27.723, 111.631, -15.124, -83.255, 50.815]
  Call Extruder(0.055)
  MoveL 6281 to (500.34, 492.3, 13.3) mm, rotated rx 0 ry 90 rz 0 deg; joints [-11.295, -27.716, 111.586, -15.302, -83.223, 50.843]
  Call Extruder(0.060)
  MoveL 6282 to (502.42, 492.3, 13.3) mm, rotated rx 0 ry 90 rz 0 deg; joints [-11.257, -27.678, 111.338, -15.27, -83.02, 50.895]
  Call Extruder(0.007)
  MoveL 6283 to (502.77, 492.3, 13.3) mm, rotated rx 0 ry 90 rz 0 deg; joints [-11.251, -27.671, 111.296, -15.265, -82.985, 50.903]
  Set speed (120.0 mm/s)
  MoveL 6284 to (502.77, 491.95, 13.3) mm, rotated rx 0 ry 90 rz 0 deg; joints [-11.218, -27.672, 111.304, -15.232, -82.991, 50.898]
  Set speed (1000.0 mm/s)
  MoveL 6285 to (502.77, 491.9, 13.3) mm, rotated rx 0 ry 90 rz 0 deg; joints [-11.214, -27.673, 111.305, -15.228, -82.992, 50.897]
  Set speed (1000.0 mm/s)
  MoveL 6286 to (503.47, 491.9, 13.3) mm, rotated rx 0 ry 90 rz 0 deg; joints [-11.201, -27.66, 111.221, -15.217, -82.924, 50.915]
  Set speed (1000.0 mm/s)
  MoveL 6287 to (496.37, 492.33, 13.3) mm, rotated rx 0 ry 90 rz 0 deg; joints [-11.371, -27.788, 112.06, -15.366, -83.613, 50.744]
  Set speed (1000.0 mm/s)
  MoveL 6288 to (490.68, 490.68, 13.3) mm, rotated rx 0 ry 90 rz 0 deg; joints [-11.324, -27.891, 112.774, -15.301, -84.201, 50.577]
  Set speed (1000.0 mm/s)
  MoveL 6289 to (490.68, 490.68, 13.4) mm, rotated rx 0 ry 90 rz 0 deg; joints [-11.324, -27.901, 112.779, -15.302, -84.196, 50.578]
  Set speed (30.0 mm/s)
  Call Extruder(0.767)
  MoveL 6290 to (509.32, 509.32, 13.4) mm, rotated rx 0 ry 90 rz 0 deg; joints [-12.669, -27.483, 110.082, -16.731, -82.046, 51.354]
  MoveL 6291 to (509.44, 509.44, 13.4) mm, rotated rx 0 ry 90 rz 0 deg; joints [-12.677, -27.48, 110.064, -16.741, -82.032, 51.359]
  Set speed (120.0 mm/s)
  MoveL 6292 to (507.39, 502.51, 13.4) mm, rotated rx 0 ry 90 rz 0 deg; joints [-12.094, -27.552, 110.494, -16.138, -82.355, 51.185]
  Set speed (30.0 mm/s)
  Call Extruder(0.280)
  MoveL 6293 to (500.58, 509.32, 13.4) mm, rotated rx 0 ry 90 rz 0 deg; joints [-12.847, -27.655, 111.129, -16.878, -82.891, 51.119]
  Set speed (120.0 mm/s)
  MoveL 6294 to (499.42, 509.32, 13.4) mm, rotated rx 0 ry 90 rz 0 deg; joints [-12.872, -27.676, 111.267, -16.898, -83.003, 51.088]
  Set speed (30.0 mm/s)
  Call Extruder(0.360)
  MoveL 6295 to (490.68, 500.58, 13.4) mm, rotated rx 0 ry 90 rz 0 deg; joints [-12.247, -27.867, 112.535, -16.235, -84.017, 50.717]
  Set speed (120.0 mm/s)
  MoveL 6296 to (490.68, 499.42, 13.4) mm, rotated rx 0 ry 90 rz 0 deg; joints [-12.139, -27.871, 112.564, -16.126, -84.039, 50.7]
  Set speed (30.0 mm/s)
  Call Extruder(0.281)
  MoveL 6297 to (497.52, 492.58, 13.4) mm, rotated rx 0 ry 90 rz 0 deg; joints [-11.373, -27.777, 111.922, -15.372, -83.491, 50.778]
  MoveL 6298 to (497.64, 492.46, 13.4) mm, rotated rx 0 ry 90 rz 0 deg; joints [-11.36, -27.775, 111.91, -15.358, -83.481, 50.779]
  Set speed (120.0 mm/s)
  MoveL 6299 to (499.08, 491.02, 13.4) mm, rotated rx 0 ry 90 rz 0 deg; joints [-11.201, -27.754, 111.773, -15.202, -83.364, 50.794]
  Set speed (30.0 mm/s)
  Call Extruder(0.014)
  MoveL 6300 to (499.42, 490.68, 13.4) mm, rotated rx 0 ry 90 rz 0 deg; joints [-11.163, -27.749, 111.74, -15.165, -83.336, 50.797]
  Set speed (120.0 mm/s)
  MoveL 6301 to (500.38, 492.33, 13.4) mm, rotated rx 0 ry 90 rz 0 deg; joints [-11.297, -27.726, 111.586, -15.304, -83.214, 50.846]
  Set speed (1000.0 mm/s)
  MoveL 6302 to (502.48, 492.58, 13.4) mm, rotated rx 0 ry 90 rz 0 deg; joints [-11.282, -27.686, 111.329, -15.295, -83.004, 50.902]
  Set speed (30.0 mm/s)
  Call Extruder(0.202)
  MoveL 6303 to (507.39, 497.49, 13.4) mm, rotated rx 0 ry 90 rz 0 deg; joints [-11.639, -27.573, 110.62, -15.675, -82.441, 51.102]
  MoveL 6304 to (507.51, 497.61, 13.4) mm, rotated rx 0 ry 90 rz 0 deg; joints [-11.648, -27.57, 110.603, -15.685, -82.427, 51.107]
  Set speed (120.0 mm/s)
  MoveL 6305 to (508.58, 498.68, 13.4) mm, rotated rx 0 ry 90 rz 0 deg; joints [-11.724, -27.544, 110.447, -15.767, -82.305, 51.152]
  Set speed (30.0 mm/s)
  Call Extruder(0.030)
  MoveL 6306 to (509.32, 499.42, 13.4) mm, rotated rx 0 ry 90 rz 0 deg; joints [-11.777, -27.527, 110.34, -15.824, -82.221, 51.183]
  Set speed (120.0 mm/s)
  MoveL 6307 to (507.64, 498.43, 13.4) mm, rotated rx 0 ry 90 rz 0 deg; joints [-11.719, -27.564, 110.567, -15.758, -82.401, 51.124]
  Set speed (1000.0 mm/s)
  MoveL 6308 to (507.64, 495.87, 13.4) mm, rotated rx 0 ry 90 rz 0 deg; joints [-11.487, -27.574, 110.63, -15.522, -82.444, 51.082]
  Set speed (1000.0 mm/s)
  MoveL 6309 to (509.32, 490.68, 13.4) mm, rotated rx 0 ry 90 rz 0 deg; joints [-10.985, -27.562, 110.552, -15.019, -82.365, 51.04]
  Set speed (30.0 mm/s)
  Call Extruder(0.767)
  MoveL 6310 to (490.68, 509.32, 13.4) mm, rotated rx 0 ry 90 rz 0 deg; joints [-13.056, -27.833, 112.303, -17.054, -83.849, 50.848]
  MoveL 6311 to (490.56, 509.44, 13.4) mm, rotated rx 0 ry 90 rz 0 deg; joints [-13.07, -27.835, 112.314, -17.068, -83.859, 50.846]
  Set speed (120.0 mm/s)
  MoveL 6312 to (502.91, 492.37, 13.4) mm, rotated rx 0 ry 90 rz 0 deg; joints [-11.255, -27.679, 111.283, -15.269, -82.966, 50.909]
  Set speed (1000.0 mm/s)
  MoveL 6313 to (502.84, 492.3, 13.4) mm, rotated rx 0 ry 90 rz 0 deg; joints [-11.249, -27.681, 111.293, -15.264, -82.974, 50.906]
  Set speed (15.0 mm/s)
  Call Extruder(0.010)
  MoveL 6314 to (502.84, 491.95, 13.4) mm, rotated rx 0 ry 90 rz 0 deg; joints [-11.217, -27.682, 111.302, -15.231, -82.98, 50.901]
  Call Extruder(0.035)
  MoveL 6315 to (502.83, 490.75, 13.4) mm, rotated rx 0 ry 90 rz 0 deg; joints [-11.107, -27.686, 111.33, -15.12, -83, 50.883]
  Call Extruder(0.010)
  MoveL 6316 to (502.83, 490.4, 13.4) mm, rotated rx 0 ry 90 rz 0 deg; joints [-11.075, -27.688, 111.338, -15.087, -83.006, 50.878]
  Call Extruder(0.007)
  MoveL 6317 to (503.18, 490.4, 13.4) mm, rotated rx 0 ry 90 rz 0 deg; joints [-11.069, -27.681, 111.297, -15.082, -82.971, 50.886]
  Call Extruder(0.187)
  MoveL 6318 to (509.6, 490.4, 13.4) mm, rotated rx 0 ry 90 rz 0 deg; joints [-10.955, -27.557, 110.525, -14.989, -82.342, 51.043]
  Call Extruder(0.160)
  MoveL 6319 to (509.6, 495.9, 13.4) mm, rotated rx 0 ry 90 rz 0 deg; joints [-11.453, -27.535, 110.393, -15.495, -82.253, 51.132]
  Call Extruder(0.056)
  MoveL 6320 to (507.67, 495.9, 13.4) mm, rotated rx 0 ry 90 rz 0 deg; joints [-11.489, -27.574, 110.626, -15.524, -82.441, 51.084]
  Call Extruder(0.063)
  MoveL 6321 to (507.67, 498.05, 13.4) mm, rotated rx 0 ry 90 rz 0 deg; joints [-11.684, -27.565, 110.573, -15.723, -82.404, 51.119]
  Call Extruder(0.010)
  MoveL 6322 to (507.67, 498.4, 13.4) mm, rotated rx 0 ry 90 rz 0 deg; joints [-11.716, -27.564, 110.564, -15.755, -82.398, 51.124]
  Call Extruder(0.007)
  MoveL 6323 to (508.02, 498.4, 13.4) mm, rotated rx 0 ry 90 rz 0 deg; joints [-11.71, -27.557, 110.522, -15.75, -82.364, 51.133]
  Call Extruder(0.036)
  MoveL 6324 to (509.25, 498.4, 13.4) mm, rotated rx 0 ry 90 rz 0 deg; joints [-11.686, -27.532, 110.374, -15.731, -82.245, 51.164]
  Call Extruder(0.010)
  MoveL 6325 to (509.6, 498.4, 13.4) mm, rotated rx 0 ry 90 rz 0 deg; joints [-11.68, -27.525, 110.332, -15.726, -82.211, 51.173]
  Call Extruder(0.007)
  MoveL 6326 to (509.6, 498.75, 13.4) mm, rotated rx 0 ry 90 rz 0 deg; joints [-11.712, -27.524, 110.323, -15.758, -82.205, 51.179]
  Call Extruder(0.046)
  MoveL 6327 to (509.6, 500.34, 13.4) mm, rotated rx 0 ry 90 rz 0 deg; joints [-11.855, -27.517, 110.283, -15.904, -82.178, 51.206]
  Call Extruder(0.010)
  MoveL 6328 to (509.6, 500.69, 13.4) mm, rotated rx 0 ry 90 rz 0 deg; joints [-11.887, -27.516, 110.274, -15.936, -82.172, 51.212]
  Call Extruder(0.007)
  MoveL 6329 to (509.25, 500.69, 13.4) mm, rotated rx 0 ry 90 rz 0 deg; joints [-11.893, -27.523, 110.316, -15.942, -82.206, 51.203]
  Call Extruder(0.036)
  MoveL 6330 to (508.02, 500.69, 13.4) mm, rotated rx 0 ry 90 rz 0 deg; joints [-11.917, -27.547, 110.464, -15.961, -82.325, 51.171]
  Call Extruder(0.010)
  MoveL 6331 to (507.67, 500.69, 13.4) mm, rotated rx 0 ry 90 rz 0 deg; joints [-11.923, -27.554, 110.507, -15.966, -82.359, 51.162]
  Call Extruder(0.007)
  MoveL 6332 to (507.67, 501.04, 13.4) mm, rotated rx 0 ry 90 rz 0 deg; joints [-11.955, -27.553, 110.498, -15.998, -82.353, 51.168]
  Call Extruder(0.062)
  MoveL 6333 to (507.67, 503.18, 13.4) mm, rotated rx 0 ry 90 rz 0 deg; joints [-12.149, -27.544, 110.443, -16.195, -82.316, 51.204]
  Call Extruder(0.056)
  MoveL 6334 to (509.6, 503.19, 13.4) mm, rotated rx 0 ry 90 rz 0 deg; joints [-12.112, -27.505, 110.21, -16.165, -82.128, 51.254]
  Call Extruder(0.187)
  MoveL 6335 to (509.6, 509.6, 13.4) mm, rotated rx 0 ry 90 rz 0 deg; joints [-12.688, -27.476, 110.04, -16.752, -82.014, 51.366]
  Call Extruder(0.559)
  MoveL 6336 to (490.4, 509.6, 13.4) mm, rotated rx 0 ry 90 rz 0 deg; joints [-13.088, -27.837, 112.328, -17.086, -83.871, 50.844]
  MoveL 6337 to (490.4, 490.4, 13.4) mm, rotated rx 0 ry 90 rz 0 deg; joints [-11.303, -27.907, 112.818, -15.28, -84.228, 50.567]
  Call Extruder(0.163)
  MoveL 6338 to (495.99, 490.4, 13.4) mm, rotated rx 0 ry 90 rz 0 deg; joints [-11.199, -27.812, 112.156, -15.191, -83.678, 50.708]
  Call Extruder(0.010)
  MoveL 6339 to (496.34, 490.4, 13.4) mm, rotated rx 0 ry 90 rz 0 deg; joints [-11.193, -27.805, 112.114, -15.186, -83.644, 50.717]
  Call Extruder(0.007)
  MoveL 6340 to (496.34, 490.75, 13.4) mm, rotated rx 0 ry 90 rz 0 deg; joints [-11.225, -27.804, 112.106, -15.219, -83.638, 50.722]
  Call Extruder(0.035)
  MoveL 6341 to (496.34, 491.95, 13.4) mm, rotated rx 0 ry 90 rz 0 deg; joints [-11.337, -27.8, 112.077, -15.331, -83.617, 50.739]
  Call Extruder(0.010)
  MoveL 6342 to (496.34, 492.3, 13.4) mm, rotated rx 0 ry 90 rz 0 deg; joints [-11.369, -27.799, 112.069, -15.364, -83.611, 50.744]
  Call Extruder(0.007)
  MoveL 6343 to (496.69, 492.3, 13.4) mm, rotated rx 0 ry 90 rz 0 deg; joints [-11.363, -27.793, 112.027, -15.359, -83.577, 50.753]
  Call Extruder(0.061)
  MoveL 6344 to (498.8, 492.3, 13.4) mm, rotated rx 0 ry 90 rz 0 deg; joints [-11.324, -27.755, 111.776, -15.326, -83.37, 50.806]
  Call Extruder(0.055)
  MoveL 6345 to (498.8, 490.4, 13.4) mm, rotated rx 0 ry 90 rz 0 deg; joints [-11.148, -27.762, 111.821, -15.148, -83.402, 50.778]
  Call Extruder(0.047)
  MoveL 6346 to (500.41, 490.4, 13.4) mm, rotated rx 0 ry 90 rz 0 deg; joints [-11.119, -27.732, 111.629, -15.124, -83.244, 50.818]
  Call Extruder(0.055)
  MoveL 6347 to (500.41, 492.3, 13.4) mm, rotated rx 0 ry 90 rz 0 deg; joints [-11.294, -27.726, 111.584, -15.301, -83.212, 50.846]
  Call Extruder(0.060)
  MoveL 6348 to (502.49, 492.3, 13.4) mm, rotated rx 0 ry 90 rz 0 deg; joints [-11.256, -27.687, 111.335, -15.269, -83.008, 50.898]
  Call Extruder(0.007)
  MoveL 6349 to (502.84, 492.3, 13.4) mm, rotated rx 0 ry 90 rz 0 deg; joints [-11.249, -27.681, 111.293, -15.264, -82.974, 50.906]
  Set speed (120.0 mm/s)
  MoveL 6350 to (502.84, 491.95, 13.4) mm, rotated rx 0 ry 90 rz 0 deg; joints [-11.217, -27.682, 111.302, -15.231, -82.98, 50.901]
  Set speed (1000.0 mm/s)
  MoveL 6351 to (502.84, 491.9, 13.4) mm, rotated rx 0 ry 90 rz 0 deg; joints [-11.213, -27.682, 111.303, -15.227, -82.981, 50.9]
  Set speed (1000.0 mm/s)
  MoveL 6352 to (503.54, 491.9, 13.4) mm, rotated rx 0 ry 90 rz 0 deg; joints [-11.2, -27.669, 111.219, -15.216, -82.912, 50.918]
  Set speed (1000.0 mm/s)
  MoveL 6353 to (496.31, 492.33, 13.4) mm, rotated rx 0 ry 90 rz 0 deg; joints [-11.372, -27.799, 112.072, -15.367, -83.614, 50.744]
  Set speed (1000.0 mm/s)
  MoveL 6354 to (490.68, 490.68, 13.4) mm, rotated rx 0 ry 90 rz 0 deg; joints [-11.324, -27.901, 112.779, -15.302, -84.196, 50.578]
  Set speed (1000.0 mm/s)
  MoveL 6355 to (490.68, 490.68, 13.5) mm, rotated rx 0 ry 90 rz 0 deg; joints [-11.324, -27.912, 112.784, -15.302, -84.191, 50.58]
